// TwinCAT 3 PLC project HeatPumpTestBenchControl
// ProgramVersion: 3.1.4022.1
// CompilerDefines: VISU_USEPROPERTYINFO
// libraries:
//   VisuElem3DPath, 3.5.6.0 (System)
//   VisuElemMeter, 3.5.6.0 (System)
//   VisuElems, 3.5.6.10 (System)
//   VisuElemsDateTime, 3.5.6.0 (System)
//   VisuElemsSpecialControls, 3.5.6.0 (System)
//   VisuElemsWinControls, 3.5.6.0 (System)
//   VisuElemTextEditor, 3.5.6.0 (System)
//   visuinputs, 3.5.6.0 (system)
//   VisuNativeControl, 3.5.6.0 (System)
//   Tc2_Standard, * (Beckhoff Automation GmbH)
//   Tc2_System, * (Beckhoff Automation GmbH)
//   Tc2_Utilities, * (Beckhoff Automation GmbH)
//   Tc3_Module, * (Beckhoff Automation GmbH)
//   VisuDialogs, * (System)
// project tree:
//   DUTs/ E_PowMeas.TcDUT, E_Press.TcDUT, E_TempSensVR10.TcDUT, E_TempSensPT100.TcDUT, E_IndexPowMeas.TcDUT, E_SMStatus.TcDUT (not stored), E_TempSensVR11.TcDUT (not stored), E_Terminals.TcDUT, ST_InputVar.TcDUT, ST_InputVar_PowMeas.TcDUT, ST_OutputVar.TcDUT (not stored), ST_PumpTime.TcDUT (not stored)
//   / GlobalTextList.TcGTLO, PlcTask.TcTTO (not stored), Visualization Manager.TcVMO (not stored)
//   GVLs/ DigOutputs.TcGVL (not stored), HeatingCurve.TcGVL (not stored), AnaOutputs.TcGVL, PID.TcGVL (not stored), PowMeas.TcGVL, Pressures.TcGVL, PumpTiming.TcGVL (not stored), StateMachine.TcGVL, SysCheck.TcGVL (not stored), SysCheckParams.TcGVL (not stored), TempConvDat.TcGVL (not stored), Temperatures.TcGVL (not stored), TempSetpoints.TcGVL (not stored), TerminalErrorRT.TcGVL (not stored), TimeProgs.TcGVL (not stored)
//   POUs/ CheckDivDInt.TcPOU (not stored), CheckDivLInt.TcPOU, CheckDivLReal.TcPOU, CheckDivReal.TcPOU (not stored), MAIN.TcPOU, P_GetTime.TcPOU
//   POUs/Control/ FB_AuxHeatCont.TcPOU, FB_CyclingControl.TcPOU (not stored), P_ControlMain.TcPOU
//   POUs/Control/TemperatureControl/ FB_PIDSuppTemp.TcPOU (not stored), FB_SimpleTempCont.TcPOU (not stored), F_GetTempSP.TcPOU, I_TempController.TcIO, P_SHSuppTempPID.TcPOU (not stored)
//   POUs/ErrorHandling/ F_WriteErrLog.TcPOU, P_EmShutdownAll.TcPOU, P_EmShutdownBPumpRun.TcPOU (not stored), P_EmShutdownHCPumpRun.TcPOU, P_EmShutdownPumpsRun.TcPOU, P_EmShutdownMain.TcPOU, P_ErrorHandlingMain.TcPOU, P_WriteErrLog.TcPOU
//   POUs/Initialize/ FB_InitPumpTimes.TcPOU (not stored), FB_ReadHeatCurve.TcPOU, FB_ReadNightMode.TcPOU, FB_ReadPressTab.TcPOU, FB_ReadPT100Tab.TcPOU, FB_ReadTempResTabVR11.TcPOU, P_InitMain.TcPOU (not stored), FB_ReadTempResTabVR10.TcPOU, FB_InitTimes.TcPOU
//   POUs/Read/ F_LinSens.TcPOU (not stored), F_NTCSens.TcPOU, F_PowMeasPhase.TcPOU, P_PowMeas.TcPOU (not stored), P_ReadMain.TcPOU (not stored), P_TestVals.TcPOU
//   POUs/SystemCheck/ F_CheckAmbTemp.TcPOU, F_CheckBrinePressure.TcPOU, F_CheckCompCycPress.TcPOU (not stored), F_CheckCompOutTemp.TcPOU (not stored), F_CheckHeatCirPress.TcPOU (not stored), F_CheckHeatCirTemp.TcPOU, F_CheckPhaseSeq.TcPOU, F_CheckSens.TcPOU, F_CheckTerm.TcPOU, P_SysCheckMain.TcPOU (not stored)
//   POUs/Write/ F_ConvLinAnaOutp.TcPOU, F_PumpConvPercVolt.TcPOU, FB_RampPump.TcPOU, P_WriteMain.TcPOU (not stored)
//   VISUs/ Vis_ManCont.TcVIS (not stored), StandardVis.TcVIS
// real-time tasks:
//   TASK PlcTask: cycle T#10ms, priority 20, ADS port 350
// I/O:
//   DEVICE Device 1 (EtherCAT) (disabled), AmsNetId 134.61.132.51.2.1
//     Coupler (EK1100) [EK1100 EtherCAT Coupler (2A E-Bus)]
//       InpPressSens (EL3064) [EL3064 4Ch. Ana. Input 0-10V]
//       InpTempSens1 (EL3204-0200) [EL3204-0200 4Ch. Ana. In. PT1000 (RTD)]
//       InpTempSens2 (EL3204-0200) [EL3204-0200 4Ch. Ana. In. PT1000 (RTD)]
//       InpTempSens3 (EL3204-0200) [EL3204-0200 4Ch. Ana. In. PT1000 (RTD)]
//       InpPowMeas (EL3403-0010) [EL3403-0010 3Ch. Power Measuring, 5A]
//       AnalogOutp (EL4004) [EL4004 4Ch. Ana. Output 0-10V, 12bit]
//       OutpSwitchValv (EL2652) [EL2652 2Ch. Relay Output, CO (230V AC / 30V DC)]
//       OutpCont (EL2622) [EL2622 2Ch. Relay Output, NO (230V AC / 30V DC)]
//       InpTempSens3wire (EL3214) [EL3214 4Ch. Ana. Input PT100 (RTD)]

// ---- DUTs/E_PowMeas.TcDUT
TYPE E_PowMeas :
(
	L1,	//power phase 1
	L2,	//power phase 2
	L3	//power phase 3
);
END_TYPE

// ---- DUTs/E_Press.TcDUT
TYPE E_Press :
(
	HP,		//High pressure - after compression
	LP,		//Low pressure	- before compression
	HCP,	//Heating circuit pressure
	BP		//Brine circuit pressure
);
END_TYPE

// ---- DUTs/E_TempSensVR10.TcDUT
TYPE E_TempSensVR10 : //all VR10 temperature sensors
(
	SP,		//Temperature of DHW storage tank
	VF1,	//Temperature at the top of the space heating buffer tank
	VF2,	//Temperature after external mixing valve
	RF1		//Temperature at the bottom of the space heating buffer tank
);
END_TYPE

// ---- DUTs/E_TempSensPT100.TcDUT
TYPE E_TempSensPT100 :
(
	TExpVEv,	//Temperature between expansion valve and evaporator
	TShEv,		//Temperature after evaporator
	TCond,		//Temperature after condenser
	TAmb		//Ambient temperature
);
END_TYPE

// ---- DUTs/E_IndexPowMeas.TcDUT
TYPE E_IndexPowMeas :
//Index-value connection of the second output of the power measurement terminal
(ApparantPower, ReactivePower, Energy, cosPhi, Frequency, negEnergy);
END_TYPE

// ---- DUTs/E_Terminals.TcDUT
TYPE E_Terminals :
(
	TempSens1,
	TempSens2,
	TempSens3,
	TempSens3Wire,
	PressSens,
	PowMeasTerm,
	AnalogOutp,
	OutpSwitchValv,
	OutpCont
);
END_TYPE

// ---- DUTs/ST_InputVar.TcDUT
TYPE ST_InputVar :
STRUCT
	(*
fVar = nVarInput*fParaM + fParaC

fParaMinVal<=fVal<=fParaMaxVal
	*)	
	
	//Raw input from terminal
	nVarInput	AT %I*	:DINT; 		//Integer input from terminal
	bSensErr	AT %I*	:BOOL;		//Sensor error bit
	
	//Physical value
	fVal				:REAL;		//Input value as REAL/FLOAT/SINGLE
	
	//Linear conversion factors
	fParaM				:REAL; 		//slope of linear conversion
	fParaC				:REAL;		//offset of linear conversion
	
	//Physical limits
	fParaMaxVal			:REAL;		//Maximum physical value
	fParaMinVal			:REAL;		//Minimum physical value
	
	bValid				:BOOL	:=	TRUE;	//Indicator if fVal is valid
	
END_STRUCT
END_TYPE

// ---- DUTs/ST_InputVar_PowMeas.TcDUT
TYPE ST_InputVar_PowMeas :
STRUCT
	//Input from terminal as INT32
	nCurrentRaw	AT	%I*	:	DINT;
	nVoltRaw	AT	%I*	:	DINT;
	nEffPowRaw	AT	%I*	:	DINT;
	nVariantRaw	AT	%I*	:	DINT;				//set to cos(phi)
(*
variant input is controlled by index output:
0	-	Apparent power
1	-	Reactive power
2	-	Energy
3	-	cos(phi)
4	-	Frequency
5	-	Negative Energy
*)	
	//Index output to terminal
	nIndexOut	AT	%Q*	:	USINT	:=	3;		//cos(phi)
	
	//Physical values
	fCurrent	:	REAL;
	fVolt		:	REAL;
	fEffPow		:	REAL;
	fcosPhi		:	REAL;
	
	//Conversion factors
	fScaleCurr		:	REAL	:=	0.000005;	//Current = 0.000005A * current transformer ratio * raw value
	fScaleVolt		:	REAL	:=	0.0001;		//Voltage = 0.0001V * voltage transformer ratio * raw value
	fScaleEffPow	:	REAL	:=	0.01;		//EffPow = 0.01W * current and voltage transformer ratio
	fCurrTrans		:	REAL	:=	0.1; 		//current transformer ratio: A50/A5
	fScaleAppPow	:	REAL	:=	0.01;		//AppPow = 0.01W * current and voltage transformer ratio * raw value
	fScaleReaPow	:	REAL	:=	0.01;		//ReaPow = 0.01VAr * current and voltage transformer ratio * raw value
	fScaleEn		:	REAL	:=	0.001;		//Energy = 0.001Wh * current and voltage transformer ratio * raw value
	fScaleCosPhi	:	REAL	:=	0.001;		//CosPhi = 0.001 * raw value
	fScaleFrequ		:	REAL	:=	0.1;		//Frequ = 0.1Hz * raw value
		
END_STRUCT
END_TYPE

// ---- GVLs/AnaOutputs.TcGVL
{attribute 'qualified_only'}
VAR_GLOBAL
	stOutpBP		:	ST_OutputVar;	//Control signal for brine pump
	stOutpIntHP		:	ST_OutputVar;	//Control signal for internal heating circuit pump
	stOutpExtHP		:	ST_OutputVar;	//Control signal for external heating circuit pump
	stOutpMixValv	:	ST_OutputVar;	//Control signal for circulating pump
END_VAR

// ---- GVLs/PowMeas.TcGVL
VAR_GLOBAL
	//Power measurement values for all phases
	ePowMeas	:	E_PowMeas;
	stPowMeas	:	ARRAY[0..2]	OF ST_InputVar_PowMeas;
	
	//accumulated values
	fEffPow		:	REAL;	//Total effective power = sum of effective power of phases
	fMeanCosPhi	:	REAL;	//Mean power factor
	fAppPow		:	REAL;	//Total apparent power
	fReaPow		:	REAL;	//Total reactive power
	
	//phase sequence
	bPhaseSeq	AT	%I*	: BOOL;	//Phase sequence detected by the power measurement terminal
	//0 - Sequence L1-L3-L2 detected -> counter-clockwise net
	//1 - Sequence L1-L2-L3 detected -> clockwise net, or at least 1 wire not connected
	
END_VAR

// ---- GVLs/Pressures.TcGVL
{attribute 'qualified_only'}
VAR_GLOBAL
	ePress	:	E_Press;
	stPress	:	ARRAY[0..3] OF ST_InputVar;

(*
	stHP	:	ST_InputVar;	//High pressure - after compression
	stLP	: 	ST_InputVar;	//Low pressure	- before compression
	stHCP	:	ST_InputVar;	//Heating circuit pressure
	stBP	:	ST_InputVar;	//Brine circuit pressure
*)
END_VAR

// ---- GVLs/StateMachine.TcGVL
{attribute 'qualified_only'}
VAR_GLOBAL
	eStatus			:	E_SMStatus	:= Initialize;
	dtCurTime		:	DT;
	todCurTime		:	TOD;
	bActAuxHeat		:	BOOL	:= TRUE;	//Activate auxiliary heater
	//Fault status
	bFault			:	BOOL	:= FALSE;	//system fault indicator
	nFault			:	USINT;				//fault number
	sFaultMess		:	STRING	:= '';		//fault message
	nErrCount		:	INT		:= 0;		//error counter
	bPermShut		:	BOOL	:= FALSE;	//permanent shutdown
	bTempShut		:	BOOL	:= FALSE;	//temporary shutdown
	bEmOpPoss		:	BOOL	:= FALSE;	//emergency operation possible
	bEmOpAct		:	BOOL	:= FALSE;	//emergency operation active
	bManEmShutdown	:	BOOL	:= FALSE;	//manual emergency shutdown
	//Cycling control
	dtLastStart		:	DT;					//date and time of last start
	dtLastStop		:	DT;					//date and time of last stop
	nNumStart		:	USINT	:= 0;		//number of starts per hour
	//Control signals
	bCompRun		:	BOOL;
	bAuxHeatOp		:	BOOL;
	bSwitchVal		:	BOOL;				//True: space heating mode || False: DHW mode
	fMixVal			:	REAL;				//mixing valve position [0..10V]
	bBrinePump		:	BOOL;
	nBrinePump		:	USINT	:= 100;		//brine pump rpm in percent (0% - minimum speed, 100% - maximum speed)
	bIntHeatCPump	:	BOOL;
	nIntHeatCPump	:	USINT	:= 100;		//internal heating circuit pump rpm in percent (0% - minimum speed, 100% - maximum speed)
	bExtHeatCPump	:	BOOL;
	nExtHeatCPump	:	USINT	:= 100;		//external heating circuit pump rpm in percent (0% - minimum speed, 100% - maximum speed)
	bCircPump		:	BOOL;
END_VAR

// ---- POUs/Control/TemperatureControl/I_TempController.TcIO
INTERFACE I_TempController

//request compressor operation

//Switching valve mode: 
//True: space heating mode
//False: DHW mode

PROPERTY CompOp : BOOL
GET
END_GET
SET
END_SET
END_PROPERTY

PROPERTY SpaceHeatTempSP : REAL
GET
END_GET
SET
END_SET
END_PROPERTY

PROPERTY ValveMode : BOOL
GET
END_GET
SET
END_SET
END_PROPERTY

END_INTERFACE

// ---- POUs/CheckDivLInt.TcPOU
// Implicitly generated code : DO NOT EDIT
FUNCTION CheckDivLInt : LINT
VAR_INPUT
	divisor:LINT;
END_VAR

// Implicitly generated code : Only an Implementation suggestion
IF divisor = 0 THEN
	CheckDivLInt:=1;
	StateMachine.bFault		:=	TRUE;
	StateMachine.nFault		:=	2;
	StateMachine.sFaultMess	:=	'Critical program error: division by 0';
	StateMachine.eStatus	:=	Error;
	P_EmShutdownAll();	//Execute emergency shutdown
ELSE
	CheckDivLInt:=divisor;
END_IF;

END_FUNCTION

// ---- POUs/ErrorHandling/P_EmShutdownAll.TcPOU
PROGRAM P_EmShutdownAll
VAR
END_VAR

//shut down all components

StateMachine.bCompRun		:=	FALSE;
DigOutputs.bOutpComp		:=	FALSE;

StateMachine.bAuxHeatOp		:=	FALSE;
DigOutputs.bOutpAH			:=	FALSE;

StateMachine.bBrinePump		:=	FALSE;
AnaOutputs.stOutpBP.fVal	:=	0.75;	//0.75 Volt: Pump stop
AnaOutputs.stOutpBP			:=	F_ConvLinAnaOutp(stOutput:=AnaOutputs.stOutpBP);

StateMachine.bIntHeatCPump	:=	FALSE;
AnaOutputs.stOutpIntHP.fVal	:=	0.75;	//0.75 Volt: Pump stop
AnaOutputs.stOutpIntHP		:=	F_ConvLinAnaOutp(stOutput:=AnaOutputs.stOutpIntHP);

StateMachine.bExtHeatCPump	:=	FALSE;
AnaOutputs.stOutpExtHP.fVal	:=	0.75;	//0.75 Volt: Pump stop
AnaOutputs.stOutpExtHP			:=	F_ConvLinAnaOutp(stOutput:=AnaOutputs.stOutpExtHP);

StateMachine.bCircPump		:=	FALSE;

END_PROGRAM

// ---- POUs/Write/F_ConvLinAnaOutp.TcPOU
FUNCTION F_ConvLinAnaOutp : ST_OutputVar
VAR_INPUT
	stOutput	:	ST_OutputVar;
END_VAR
VAR
END_VAR

//nVarOutput = (fVar-fParaC)/fParaM)
stOutput.nVarOutput	:=	REAL_TO_INT((stOutput.fVal - stOutput.fParaC)*stOutput.fParaMaxOutp/stOutput.nParaMaxInt);

//assign output
F_ConvLinAnaOutp	:=	stOutput;

END_FUNCTION

// ---- POUs/CheckDivLReal.TcPOU
// Implicitly generated code : DO NOT EDIT
FUNCTION CheckDivLReal : LREAL
VAR_INPUT
	divisor:LREAL;
END_VAR

// Implicitly generated code : Only an Implementation suggestion
IF divisor = 0 THEN
	CheckDivLReal:=1;
	StateMachine.bFault		:=	TRUE;
	StateMachine.nFault		:=	2;
	StateMachine.sFaultMess	:=	'Critical program error: division by 0';
	StateMachine.eStatus	:=	Error;
	P_EmShutdownAll();	//Execute emergency shutdown
ELSE
	CheckDivLReal:=divisor;
END_IF;

END_FUNCTION

// ---- POUs/Control/FB_AuxHeatCont.TcPOU
FUNCTION_BLOCK FB_AuxHeatCont
VAR_INPUT
	bCompOp			:	BOOL	:=	FALSE; //has the controller requested compressor operation
	bCycContOK		:	BOOL; //has the cycling control authorized the compressor start-up
	bCompStart		:	BOOL; //is compressor start-up procedure active
END_VAR
VAR_OUTPUT
	bAuxHeatOp	:	BOOL;
END_VAR
VAR
	eVF1	:	E_TempSensVR10	:=	VF1;
	eSP		:	E_TempSensVR10	:=	SP;
	SampTim	:	TON();						//Sampling timer
	fBuffVF1:	ARRAY[0..nAuxHeatStart] OF REAL;	//Buffer
	fBuffSP	:	ARRAY[0..nAuxHeatStart] OF REAL;	//Buffer
	i		:	INT;
	bAuxCap	:	BOOL;
END_VAR
VAR CONSTANT
	nAuxHeatStart	:	INT		:=	180;	//Time in seconds the auxiliary heater control waits for the heat pump to be effective
END_VAR

IF bCompOp AND (NOT bAuxHeatOp) AND bCycContOK THEN

	SampTim.IN	:=	TRUE;
	SampTim.PT	:=	T#1s;
	SampTim();

	IF SampTim.Q THEN
		FOR i := 0 TO nAuxHeatStart - 1 DO
			fBuffVF1[i]	:=	fBuffVF1[i+1];
		END_FOR
		fBuffVF1[nAuxHeatStart] := Temperatures.stTempSensVR10[eVF1].fVal; //save current temperature in buffer
	
		FOR i := 0 TO nAuxHeatStart - 1 DO
			fBuffSP[i]	:=	fBuffSP[i+1];
		END_FOR
		fBuffSP[nAuxHeatStart] := Temperatures.stTempSensVR10[eSP].fVal; //save current temperature in buffer
	
		//reset timer
		SampTim.IN	:=	FALSE;
		SampTim();
	END_IF
	
	//check if auxiliary heater is needed
	IF StateMachine.bSwitchVal THEN	//space heating mode
		IF (fBuffVF1[nAuxHeatStart] < fBuffVF1[0]) THEN //temperature in buffer tank has not increased
			bAuxHeatOp	:=	TRUE;	//activate auxiliary heater
			bAuxCap		:=	TRUE;
		END_IF
	ELSE	//DHW mode
		IF (fBuffSP[nAuxHeatStart] < fBuffSP[0]) THEN //temperature in buffer tank has not increased
			bAuxHeatOp	:=	TRUE;	//activate auxiliary heater
			bAuxCap		:=	TRUE;
		END_IF
	END_IF
ELSIF bCompOp AND  (NOT bAuxHeatOp) AND (NOT bCycContOK) THEN	//heat demand, but compressor cannot start
	bAuxHeatOp	:=	TRUE;	
ELSIF (NOT bCompOp) THEN	//deactivate auxiliary heater when no compressor operation is needed
	bAuxHeatOp	:=	FALSE;
	bAuxCap 	:=	FALSE;
ELSIF bAuxHeatOp AND bCycContOK AND (NOT bAuxCap) AND NOT (bCompStart) THEN //deactivate auxiliary heater when the compressor can start again
	bAuxHeatOp := FALSE;
END_IF

END_FUNCTION_BLOCK

// ---- POUs/Control/P_ControlMain.TcPOU
PROGRAM P_ControlMain
VAR_INPUT
	bEmOp				:	BOOL	:=	FALSE;	//Emergency operation
END_VAR
VAR
	iTempCont			:	I_TempController;	//temperature controller interface
	//function block instances
	fbSimpleTempCont	:	FB_SimpleTempCont;	//temperature controller
	fbCycCont			:	FB_CyclingControl;
	fbAuxHeatCont		:	FB_AuxHeatCont;		//auxiliary heater control
	
	//compressor startup and shutdown flags
	bCompStart				:	BOOL	:= FALSE;
	bCompStop				:	BOOL	:= FALSE;
	bShutdownPump			:	BOOL	:= FALSE;
	bShutdownPumpAux		:	BOOL;
	bAuxHeatOld				:	BOOL;
	
	//pump timing
	TimBP					:	TON;
	TimIntHeatCir			:	TON;
	TimIntHeatCirAux		:	TON;
	TimIntHeatCirEm			:	TON;
END_VAR

//These lines need to be adjusted to use a different controller
fbSimpleTempCont();					//execute temperature control function block
iTempCont	:=	fbSimpleTempCont;	//assign function block to interface

//set switching valve mode
StateMachine.bSwitchVal	:=	iTempCont.ValveMode;

//read space heating temperature setpoint
TempSetpoints.fSpaceHeatSP	:=	iTempCont.SpaceHeatTempSP;

IF (NOT bEmOp) THEN //normal operation
	
	//operate circulating pump
	IF (TOD_TO_DINT(StateMachine.todCurTime) > TOD_TO_DINT(TimeProgs.todNightModeEnd)) AND
		(TOD_TO_DINT(StateMachine.todCurTime) < TOD_TO_DINT(TimeProgs.todNightModeStart)) THEN //day
		StateMachine.bCircPump	:=	TRUE;
	ELSE
		StateMachine.bCircPump	:=	FALSE;
	END_IF

	IF iTempCont.CompOp AND (NOT StateMachine.bCompRun) THEN	//compressor operation requested by controller and compressor not already running
		//execute cycling control
		fbCycCont();
		IF (NOT StateMachine.bFault) AND fbCycCont.bStartupOK THEN	//system is not in fault state and cycling OK
			bCompStart	:=	TRUE;		//give compressor start signal
		END_IF
	ELSIF (NOT iTempCont.CompOp) AND StateMachine.bCompRun THEN	//no compressor operation requested by controller and compressor running
		//execute cycling control
		fbCycCont();
		IF fbCycCont.bShutdownOK THEN
			bCompStop	:= TRUE;
		END_IF
	END_IF

	//compressor startup procedure
	IF bCompStart THEN
		//start pumps
		IF PumpTiming.stBPTime.bFirst THEN					//brine pump first
			StateMachine.bBrinePump	:=	TRUE;
			TimBP.PT				:=	PumpTiming.stBPTime.tPre;
			TimBP.IN				:=	TRUE;
			TimIntHeatCir.PT		:=	PumpTiming.stIntHeatCirTime.tDelay;
			TimIntHeatCir.IN		:=	TRUE;
			TimBP();
			TimIntHeatCir();
			IF TimIntHeatCir.Q THEN
				StateMachine.bIntHeatCPump	:=	TRUE;
			END_IF
		ELSIF PumpTiming.stIntHeatCirTime.bFirst THEN		//internal heating circuit pump first
			StateMachine.bIntHeatCPump	:=	TRUE;
			TimIntHeatCir.PT			:=	PumpTiming.stIntHeatCirTime.tPre;
			TimIntHeatCir.IN			:=	TRUE;
			TimBP.PT					:=	PumpTiming.stBPTime.tDelay;
			TimBP.IN					:=	TRUE;
			TimIntHeatCir();
			TimBP();
			IF TimBP.Q THEN
				StateMachine.bBrinePump		:=	TRUE;
			END_IF
		END_IF
	
		//start compressor
		IF TimBP.Q AND TimIntHeatCir.Q THEN
			//reset timers
			TimBP.IN					:=	FALSE;
			TimIntHeatCir.IN			:=	FALSE;
			TimBP();
			TimIntHeatCir();
		
			StateMachine.dtLastStart	:=	StateMachine.dtCurTime;
			StateMachine.nNumStart		:=	StateMachine.nNumStart + 1;	//startup counter
			StateMachine.bCompRun		:=	TRUE;
			bCompStart					:=	FALSE;						//startup complete
		END_IF
	END_IF

	//compressor shutdown procedure
	IF bCompStop THEN
		StateMachine.dtLastStop		:=	StateMachine.dtCurTime;
		StateMachine.bCompRun		:=	FALSE;
		bShutdownPump				:=	TRUE;
		bCompStop					:=	FALSE;
	END_IF

	IF bShutDownPump THEN
		//pump timing
		TimBP.PT					:=	PumpTiming.stBPTime.tPost;
		TimBP.IN					:=	TRUE;
		TimIntHeatCir.PT			:=	PumpTiming.stIntHeatCirTime.tPost;
		TimIntHeatCir.IN			:=	TRUE;
		TimBP();
		TimIntHeatCir();
		IF TimBP.Q THEN	//stop brine pump
			TimBP.IN				:=	FALSE;
			StateMachine.bBrinePump	:=	FALSE;
		END_IF
		IF TimIntHeatCir.Q THEN	//stop internal heating circuit pump
			TimIntHeatCir.IN			:=	FALSE;
			StateMachine.bIntHeatCPump	:=	FALSE;
		END_IF
		IF TimIntHeatCir.Q AND TimBP.Q THEN
			TimBP();
			TimIntHeatCir();
			bShutDownPump				:=	FALSE;	//shutdown complete
		END_IF
	END_IF
	TimIntHeatCirEm(IN:=FALSE); //reset emergency operation timer
ELSE	//emergency operation
	StateMachine.bCompRun		:=	FALSE;
	StateMachine.bBrinePump		:=	FALSE;
	StateMachine.bIntHeatCPump	:=	TRUE;
	TimIntHeatCirEm(IN:=TRUE,PT:=PumpTiming.stIntHeatCirTime.tPre);
	StateMachine.bCircPump		:=	TRUE;
	IF iTempCont.CompOp AND TimIntHeatCirEm.Q THEN	//start auxiliary heater if temperature controller identifies demand
		StateMachine.bAuxHeatOp	:=	TRUE;
	ELSE
		StateMachine.bAuxHeatOp	:=	FALSE;
	END_IF
END_IF

//space heating supply temperature and external heating circuit pump control
P_SHSuppTempPID();

//regular auxiliary heater control
IF NOT bEmOp THEN
	IF StateMachine.bActAuxHeat THEN
		fbAuxHeatCont(bCompOp:=iTempCont.CompOp, bCycContOK:=fbCycCont.bStartupOK, bCompStart:=bCompStart);
		IF fbAuxHeatCont.bAuxHeatOp THEN			//auxiliary heater operation requested
			StateMachine.bIntHeatCPump	:=	TRUE;	//start internal heating circuit pump
			TimIntHeatCirAux(IN:=TRUE, PT:=PumpTiming.stIntHeatCirTime.tPre);
			IF TimIntHeatCirAux.Q THEN				//after 1 minute
				StateMachine.bAuxHeatOp := TRUE;	//start auxiliary heater
				TimIntHeatCirAux(In:=FALSE);		//reset timer
			END_IF
		ELSE
			StateMachine.bAuxHeatOp	:=	FALSE;
		END_IF
	ELSE
		StateMachine.bAuxHeatOp	:=	FALSE;
	END_IF
	
	IF (NOT StateMachine.bAuxHeatOp) AND bAuxHeatOld THEN	//auxiliary heater was active last cycle
		bShutdownPumpAux	:=	TRUE;
	END_IF
	
END_IF

IF bShutdownPumpAux THEN
	TimIntHeatCirAux(IN:=TRUE, PT:=PumpTiming.stIntHeatCirTime.tPost);
	IF TimIntHeatCirAux.Q THEN
		StateMachine.bIntHeatCPump	:=	FALSE;
		TimIntHeatCirAux(In:=FALSE);
		bShutdownPumpAux	:=	FALSE;
	END_IF
END_IF

bAuxHeatOld	:=	StateMachine.bAuxHeatOp;

END_PROGRAM

// ---- POUs/Control/TemperatureControl/F_GetTempSP.TcPOU
FUNCTION F_GetTempSP : REAL
VAR_INPUT
	fAmbTemp	:	REAL;	//Ambient temperature
END_VAR
VAR
	i			:	USINT	:= 0;
	nLeftInd	:	USINT;
	nRightInd	:	USINT;
	bFound		:	BOOL	:=	FALSE;	//flag if left and right element were found
	
	fDiffSet	:	REAL;				//difference between room temperature setpoint and 20°C
	fSlopeAdap	:	REAL	:=	2;		//slope of space heating setpoint adaption
	
	fIntVal		:	REAL;				//interpolated value
	fSetpoint	:	REAL;				//space heating temperature setpoint
END_VAR

FOR i:=1 TO 40 DO
	IF NOT bFound THEN
		IF HeatingCurve.HeatCurve[i,0] >= fAmbTemp THEN
			nLeftInd	:=	i - 1;
			nRightInd	:=	i;
			bFound		:=	TRUE;
		END_IF
	END_IF
END_FOR

//perform interpolation
IF bFound THEN
	fIntVal	:=	HeatingCurve.HeatCurve[nLeftInd,1] + ((HeatingCurve.HeatCurve[nRightInd,1] - HeatingCurve.HeatCurve[nLeftInd,1])/(HeatingCurve.HeatCurve[nRightInd,0] - HeatingCurve.HeatCurve[nLeftInd,0])) * (fAmbTemp - HeatingCurve.HeatCurve[nLeftInd,0]);
ELSIF HeatingCurve.HeatCurve[0,0] >= fAmbTemp THEN	//ambient temperature lower than minimum value in heating curve
	fIntVal	:=	HeatingCurve.HeatCurve[0,1];
ELSIF fAmbTemp >= HeatingCurve.HeatCurve[40,0] THEN	//ambient temperature higher than maximum value in heating curve
	fIntVal	:=	HeatingCurve.HeatCurve[40,1];
END_IF

//adapt to room temperature setpoint
IF (TOD_TO_UDINT(StateMachine.todCurTime) > TOD_TO_UDINT(TimeProgs.todNightModeEnd)) AND
	(TOD_TO_UDINT(StateMachine.todCurTime) < TOD_TO_UDINT(TimeProgs.todNightModeStart)) THEN	//day
	fDiffSet	:=	TempSetpoints.fRoomSetpoint - 20;
ELSE	//night
	fDiffSet	:=	TempSetpoints.fRoomSetpointNight - 20;
END_IF
fSetpoint	:=	fIntVal + (fDiffSet * fSlopeAdap);

//assign output
F_GetTempSP	:=	fSetpoint;

END_FUNCTION

// ---- POUs/ErrorHandling/F_WriteErrLog.TcPOU
FUNCTION F_WriteErrLog : BOOL
VAR_INPUT
END_VAR
VAR
END_VAR

END_FUNCTION

// ---- POUs/ErrorHandling/P_EmShutdownHCPumpRun.TcPOU
PROGRAM P_EmShutdownHCPumpRun
VAR
END_VAR

//shut down all components except heating circuit pumps

StateMachine.bCompRun		:=	FALSE;
DigOutputs.bOutpComp		:=	FALSE;

StateMachine.bAuxHeatOp		:=	FALSE;
DigOutputs.bOutpAH			:=	FALSE;

StateMachine.bBrinePump		:=	FALSE;
AnaOutputs.stOutpBP.fVal	:=	0.75;	//0.75 Volt: Pump stop
AnaOutputs.stOutpBP			:=	F_ConvLinAnaOutp(stOutput:=AnaOutputs.stOutpBP);

StateMachine.bIntHeatCPump	:=	TRUE;
AnaOutputs.stOutpIntHP.fVal	:=	10;
AnaOutputs.stOutpIntHP		:=	F_ConvLinAnaOutp(stOutput:=AnaOutputs.stOutpIntHP);

StateMachine.bExtHeatCPump	:=	TRUE;
AnaOutputs.stOutpExtHP.fVal	:=	10;
AnaOutputs.stOutpExtHP			:=	F_ConvLinAnaOutp(stOutput:=AnaOutputs.stOutpExtHP);

StateMachine.bCircPump		:=	TRUE;

END_PROGRAM

// ---- POUs/ErrorHandling/P_EmShutdownPumpsRun.TcPOU
PROGRAM P_EmShutdownPumpsRun
VAR
END_VAR

//shut down all components except pumps

StateMachine.bCompRun		:=	FALSE;
DigOutputs.bOutpComp		:=	FALSE;

StateMachine.bAuxHeatOp		:=	FALSE;
DigOutputs.bOutpAH			:=	FALSE;

StateMachine.bBrinePump		:=	TRUE;
AnaOutputs.stOutpBP.fVal	:=	10;
AnaOutputs.stOutpBP			:=	F_ConvLinAnaOutp(stOutput:=AnaOutputs.stOutpBP);

StateMachine.bIntHeatCPump	:=	TRUE;
AnaOutputs.stOutpIntHP.fVal	:=	10;
AnaOutputs.stOutpIntHP		:=	F_ConvLinAnaOutp(stOutput:=AnaOutputs.stOutpIntHP);

StateMachine.bExtHeatCPump	:=	TRUE;
AnaOutputs.stOutpExtHP.fVal	:=	10;
AnaOutputs.stOutpExtHP			:=	F_ConvLinAnaOutp(stOutput:=AnaOutputs.stOutpExtHP);

StateMachine.bCircPump		:=	TRUE;

END_PROGRAM

// ---- POUs/ErrorHandling/P_EmShutdownMain.TcPOU
PROGRAM P_EmShutdownMain
VAR
END_VAR

IF StateMachine.bManEmShutdown THEN
	StateMachine.bFault		:=	TRUE;
	StateMachine.nFault		:=	1;
	StateMachine.sFaultMess	:=	'Manual emergency shutdown';
END_IF

//emergency shutdown scenarios

//manual emergency shutdown or terminal communication error or initialization failed or division by 0 detected -> stop all components
IF StateMachine.bManEmShutdown OR SysCheck.bTermErrRT OR (StateMachine.nFault = 10) OR (StateMachine.nFault = 2) THEN
	P_EmShutdownAll();	//complete shutdown	
//only brine pressure fault -> keep heating circuit pump running
ELSIF (SysCheck.bBP OR (StateMachine.nFault = 54)) AND (NOT SysCheck.bHCP) THEN //brine pressure too low or sensor failure
	P_EmShutdownHCPumpRun();
//only heating circuit pressure fault -> keep brine pump running
ELSIF (SysCheck.bHCP OR (StateMachine.nFault = 53)) AND (NOT SysCheck.bBP) THEN //heating circuit pressure too low or sensor failure
	P_EmShutdownBPumpRun();
//other faults keep all pumps running
ELSE
	P_EmShutdownPumpsRun();
END_IF

END_PROGRAM

// ---- POUs/ErrorHandling/P_ErrorHandlingMain.TcPOU
PROGRAM P_ErrorHandlingMain
VAR
	HCPTim	:	TON;
	BPTim	:	TON;
END_VAR

//error handling for each fault that can occur
CASE StateMachine.nFault OF
	
	1:	//manual emergency shutdown
		StateMachine.bPermShut	:=	TRUE;
		StateMachine.bEmOpPoss	:=	FALSE;
		
	2:	//division by 0
		StateMachine.bPermShut	:=	TRUE;
		StateMachine.bEmOpPoss	:=	FALSE;
		
	10:	//Initialization failed
		StateMachine.bPermShut	:=	TRUE;
		StateMachine.bEmOpPoss	:=	FALSE;

	21:	//compressor outlet temperature too high
		StateMachine.bTempShut	:=	TRUE;	//wait for a lower temperature
		IF NOT SysCheck.bHCP THEN	//enable emergency operation if heating circuit pressure is ok
			StateMachine.bEmOpPoss	:=	TRUE;
		END_IF

	31, 32:	//heating circuit temperatures too high
		StateMachine.bTempShut	:=	TRUE;	//wait for lower temperatures
		StateMachine.bEmOpPoss	:=	FALSE;
		
	41, 42:	//ambient temperature too high or low
		StateMachine.bTempShut	:=	TRUE;	//wait for a suitable ambient temperature
		IF NOT SysCheck.bHCP THEN	//enable emergency operation if heating circuit pressure is ok
			StateMachine.bEmOpPoss	:=	TRUE;
		END_IF

	43:	//brine pressure too low
		StateMachine.bTempShut	:=	TRUE;
		IF NOT SysCheck.bHCP THEN	//enable emergency operation if heating circuit pressure is ok
			StateMachine.bEmOpPoss	:=	TRUE;
		END_IF
		BPTim.PT				:=	T#5M;
		BPTim.IN				:=	TRUE;
		BPTim();
		IF BPTim.Q THEN	//if the brine circuit pressure stays too low for 5 mins, switch to permanent shutdown
			StateMachine.bTempShut	:=	FALSE;
			StateMachine.bPermShut	:=	TRUE;
			BPTim.IN				:=	FALSE;
			BPTim();
		END_IF

	44:	//heating circuit pressure too low
		StateMachine.bTempShut	:=	TRUE;
		StateMachine.bEmOpPoss	:=	FALSE;
		HCPTim.PT				:=	T#5M;
		HCPTim.IN				:=	TRUE;
		HCPTim();
		IF HCPTim.Q THEN	//if the heating circuit pressure stays too low for 5 mins, switch to permanent shutdown
			StateMachine.bTempShut	:=	FALSE;
			StateMachine.bPermShut	:=	TRUE;
			HCPTim.IN				:=	FALSE;
			HCPTim();
		END_IF
		
	45, 46:	//evaporation pressure too low or condensation pressure too high
		StateMachine.bTempShut	:=	TRUE;
		IF NOT SysCheck.bHCP THEN	//enable emergency operation if heating circuit pressure is ok
			StateMachine.bEmOpPoss	:=	TRUE;
		END_IF

	47:	//phase sequence error
		StateMachine.bPermShut	:=	TRUE;
		IF NOT SysCheck.bHCP THEN	//enable emergency operation if heating circuit pressure is ok
			StateMachine.bEmOpPoss	:=	TRUE;
		END_IF
		
	51, 52, 54: //brine circuit pressure, high pressure or low pressure sensor failure
		StateMachine.bPermShut	:=	TRUE;
		IF NOT SysCheck.bHCP THEN	//enable emergency operation if heating circuit pressure is ok
			StateMachine.bEmOpPoss	:=	TRUE;
		END_IF
		
	53:	//heating circuit pressure sensor failure
		StateMachine.bPermShut	:=	TRUE;
		StateMachine.bEmOpPoss	:=	FALSE;	//disable emergency operation in case heating circuit pressure is too low
		
	64:	//ambient temperature sensor failure
		StateMachine.bPermShut	:=	TRUE;
		IF NOT SysCheck.bHCP THEN	//enable emergency operation if heating circuit pressure is ok
			StateMachine.bEmOpPoss	:=	TRUE;
		END_IF	
		
	71, 72, 73, 74, 75, 76, 77, 78:	//internal temperature sensor failure
		StateMachine.bPermShut	:=	TRUE;
		IF NOT SysCheck.bHCP THEN	//enable emergency operation if heating circuit pressure is ok
			StateMachine.bEmOpPoss	:=	TRUE;
		END_IF
		
	81, 82, 83, 84:	//external temperature sensor failure
		StateMachine.bPermShut	:=	TRUE;
		StateMachine.bEmOpPoss	:=	FALSE; //disable emergency operation to prevent dangerous temperatures
		
	91, 92, 93, 94, 95, 96, 97, 98, 99:	//real-time communication failure
		StateMachine.bPermShut	:=	TRUE;
		StateMachine.bEmOpPoss	:=	FALSE;

END_CASE

END_PROGRAM

// ---- POUs/ErrorHandling/P_WriteErrLog.TcPOU
PROGRAM P_WriteErrLog
VAR_INPUT
	bStart		:	BOOL;
END_VAR
VAR
	nStep		:	USINT;

	fbFileOpen	:	FB_FileOpen;
	fbFileClose	:	FB_FileClose;
	sErrLogPath	:	STRING	:=	'D:\cve-mme\WpPruefstandData\ErrorLog.txt';
	
	fbFilePuts	:	FB_FilePuts;
	sErrLogMess	:	STRING;
	
	hLogFile	:	UINT;
	nErrCount	:	INT		:=	0;
END_VAR

CASE nStep OF
	
	0:	//idle
		IF bStart THEN
			bStart	:=	FALSE;
			nStep	:=	1;
		END_IF

	1:	//open ErrorLog File
		fbFileOpen(sNetId:='', sPathName:=sErrLogPath, nMode:=FOPEN_MODEAPPEND OR FOPEN_MODEPLUS, bExecute:=TRUE);
		nStep	:=	2;
		
	2:
		IF fbFileOpen.bError THEN
			nStep	:=	0;
		END_IF
		
		IF fbFileOpen.bBusy THEN
			fbFileOpen(bExecute:=FALSE);
		ELSE
			fbFileOpen(bExecute:=FALSE);
			hLogFile	:=	fbFileOpen.hFile;
			sErrLogMess	:=	CONCAT(str1:=DT_TO_STRING(StateMachine.dtCurTime),
				str2:=CONCAT(str1:='$t',str2:=CONCAT(str1:=StateMachine.sFaultMess,str2:='$n')));
			nStep		:=	3;	
		END_IF	
		
	3:	//write data
		fbFilePuts(sNetId:='',hFile:=hLogFile,sLine:=sErrLogMess,bExecute:=TRUE);
		nStep			:=	4;
		
	4:
		IF fbFilePuts.bError THEN
			nStep	:=	0;
		END_IF
	
		IF fbFilePuts.bBusy THEN
			fbFilePuts(bExecute:=FALSE);
		ELSE
			fbFilePuts(bExecute:=FALSE);
			nStep	:=	5;
		END_IF
		
	5:	//close file
		fbFileClose(sNetId:='',hFile:=hLogFile,bExecute:=TRUE);
		nStep	:=	6;
		
	6:	
		IF fbFileClose.bError THEN
			nStep	:=	0;
		END_IF
	
		IF fbFileClose.bBusy THEN
			fbFileClose(bExecute:=FALSE);
		ELSE
			fbFileClose(bExecute:=FALSE);
			hLogFile	:=	0;
			nStep		:=	0;	//switch to idle mode
		END_IF
END_CASE

END_PROGRAM

// ---- POUs/Initialize/FB_ReadHeatCurve.TcPOU
FUNCTION_BLOCK FB_ReadHeatCurve
VAR_INPUT
	bExecute		:	BOOL	:= FALSE;
END_VAR
VAR_OUTPUT
	bCompleted		:	BOOL	:=	FALSE;
	bError			:	BOOL	:=	FALSE;
END_VAR
VAR
	fbFileOpen		:	FB_FileOpen;
	fbFileGets		:	FB_FileGets;
	fbReader		:	FB_CSVMemBufferReader;
	fbFileClose		:	FB_FileClose;
	sCSVPath		:	STRING	:=	'*\Data\HeatingCurve.csv';	//Path to csv file
	hFile			:	UINT;
	bEOF			:	BOOL	:=	FALSE;
	Step			:	DWORD	:=	0;
	sLine			:	STRING;	//Line read by fbFileGets
	nLine			:	UINT	:=	0;
END_VAR

CASE Step OF
	
0:	//Standby mode
	IF bExecute THEN
		bExecute	:=	FALSE; //reset to defaults
		hFile		:=	0;
		bEOF		:=	FALSE;
		bCompleted	:=	FALSE;
		bError		:=	FALSE;
		sLine		:=	'';
		nLine		:=	0;
		Step		:=	1; //start program
	END_IF

1:	//Open file
	fbFileOpen(sNetId:='', sPathName:=sCSVPath, nMode:=FOPEN_MODEREAD OR FOPEN_MODETEXT,
		ePath:=PATH_GENERIC, tTimeout:=T#5s, bExecute:=TRUE);
	Step	:=	Step + 1;

2:
	fbFileOpen(bExecute:=FALSE);
	IF NOT fbFileOpen.bBusy THEN
		IF NOT fbFileOpen.bError THEN
			//Store file handle
			hFile	:=	fbFileOpen.hFile;
			Step	:=	Step + 1;
		ELSE
			Step	:=	90;	
		END_IF
	END_IF

3:	//Read csv file
	fbFileGets(sNetId:='', hFile:=hFile, bExecute:=TRUE, tTimeout:=T#5S);
	nLine	:=	nLine + 1;
	Step	:=	Step + 1;

4:
	fbFileGets(bExecute:=FALSE);
	IF NOT fbFileGets.bBusy THEN
		IF NOT (nLine = 1) THEN //Header -> jump to next line
			IF NOT fbFileGets.bError THEN
				IF fbFileGets.bEOF THEN
					Step	:=	10; //Reached end of file
				ELSE
					sLine	:=	fbFileGets.sLine; //store line
					IF RIGHT(sLine,1) = '$L' THEN
						sLine	:=	REPLACE(sLINE, '$R$L', 2, LEN(sLine)); //restore CRLF characters
					END_IF
					Step	:=	Step + 1;
				END_IF
			ELSE
				Step	:=	90;
			END_IF
		ELSE
			Step	:=	3;
		END_IF
	END_IF
	
5:	//Parse line
	
	fbReader.eCmd	:=	eEnumCmd_First;	//Read first value (ambient temperature)
	fbReader(pBuffer:=ADR(sLine), cbBuffer:=SIZEOF(sLine));
	
	IF fbReader.bOk THEN
		HeatingCurve.HeatCurve[nLine-2,0] := STRING_TO_REAL(fbReader.getValue);	//account for header
	ELSE
		Step	:=	90;
	END_IF	
	
	fbReader.eCmd	:=	eEnumCmd_Next;	//Read next value (temperature setpoint)
	fbReader(pBuffer:=ADR(sLine), cbBuffer:=SIZEOF(sLine));
	
	IF fbReader.bOk THEN
		HeatingCurve.HeatCurve[nLine-2,1] := STRING_TO_REAL(fbReader.getValue); //account for header
	ELSE
		Step	:=	90;
	END_IF
	
	//Read next line
	Step	:=	3;
	
10:	//end of csv file
	IF (hFile <> 0) THEN
		Step	:=	20; //close file
	END_IF
	
20:	//close csv file
	fbFileClose(bExecute:=FALSE);
	fbFileClose(sNetId:='', hFile:=hFile, bExecute:=TRUE, tTimeout:=T#5S);
	Step	:=	21;
	
21:	
	fbFileClose(bExecute:=FALSE);
	IF NOT fbFileClose.bBusy THEN
		step	:=	0;	//Standby mode
		bCompleted	:=	TRUE;
	END_IF
	
90:	//TODO: Error handling
	bError	:=	TRUE;
	IF (hFile <> 0) THEN
		Step	:=	20;	//close file
	END_IF

END_CASE

END_FUNCTION_BLOCK

// ---- POUs/Initialize/FB_ReadNightMode.TcPOU
FUNCTION_BLOCK FB_ReadNightMode
VAR_INPUT
	bExecute		:	BOOL	:= FALSE;
END_VAR
VAR_OUTPUT
	bCompleted		:	BOOL	:=	FALSE;
	bError			:	BOOL	:=	FALSE;
END_VAR
VAR
	fbFileOpen		:	FB_FileOpen;
	fbFileGets		:	FB_FileGets;
	fbReader		:	FB_CSVMemBufferReader;
	fbFileClose		:	FB_FileClose;
	sCSVPath		:	STRING	:=	'*\Data\NightMode.csv';	//Path to csv file
	hFile			:	UINT;
	bEOF			:	BOOL	:=	FALSE;
	Step			:	DWORD	:=	0;
	sLine			:	STRING;	//Line read by fbFileGets
	nLine			:	UINT	:=	0;
	nHourStart		:	USINT;
	nHourStop		:	USINT;
	nMinStart		:	USINT;
	nMinStop		:	USINT;
	nStartTime		:	UDINT;	//Start time in ms
	nStopTime		:	UDINT;	//Stop time in ms
END_VAR

CASE Step OF
	
0:	//Standby mode
	IF bExecute THEN
		bExecute	:=	FALSE; //reset to defaults
		hFile		:=	0;
		bEOF		:=	FALSE;
		bCompleted	:=	FALSE;
		bError		:=	FALSE;
		sLine		:=	'';
		nLine		:=	0;
		Step		:=	1; //start program
	END_IF

1:	//Open file
	fbFileOpen(sNetId:='', sPathName:=sCSVPath, nMode:=FOPEN_MODEREAD OR FOPEN_MODETEXT,
		ePath:=PATH_GENERIC, tTimeout:=T#5s, bExecute:=TRUE);
	Step	:=	Step + 1;

2:
	fbFileOpen(bExecute:=FALSE);
	IF NOT fbFileOpen.bBusy THEN
		IF NOT fbFileOpen.bError THEN
			//Store file handle
			hFile	:=	fbFileOpen.hFile;
			Step	:=	Step + 1;
		ELSE
			Step	:=	90;	
		END_IF
	END_IF

3:	//Read csv file
	fbFileGets(sNetId:='', hFile:=hFile, bExecute:=TRUE, tTimeout:=T#5S);
	nLine	:=	nLine + 1;
	Step	:=	Step + 1;

4:
	fbFileGets(bExecute:=FALSE);
	IF NOT fbFileGets.bBusy THEN
		IF NOT (nLine = 1) THEN //Header -> jump to next line
			IF NOT fbFileGets.bError THEN
				IF fbFileGets.bEOF THEN
					Step	:=	10; //Reached end of file
				ELSE
					sLine	:=	fbFileGets.sLine; //store line
					IF RIGHT(sLine,1) = '$L' THEN
						sLine	:=	REPLACE(sLINE, '$R$L', 2, LEN(sLine)); //restore CRLF characters
					END_IF
					Step	:=	Step + 1;
				END_IF
			ELSE
				Step	:=	90;
			END_IF
		ELSE
			Step	:=	3;
		END_IF
	END_IF
	
5:	//Parse line
	fbReader.eCmd	:=	eEnumCmd_First;	//Read first value (identifier)
	fbReader(pBuffer:=ADR(sLine), cbBuffer:=SIZEOF(sLine));
	
	fbReader.eCmd	:=	eEnumCmd_Next;	//Read next value (hour)
	fbReader(pBuffer:=ADR(sLine), cbBuffer:=SIZEOF(sLine));
	
	IF fbReader.bOk THEN
		IF (nLine = 2) THEN
			nHourStart	:=	STRING_TO_USINT(fbReader.getValue);
		ELSIF (nLine = 3) THEN
			nHourStop	:=	STRING_TO_USINT(fbReader.getValue);
		ELSE
			Step	:=	90;
		END_IF
	ELSE
		Step	:=	90;
	END_IF	
	
	fbReader.eCmd	:=	eEnumCmd_Next;	//Read next value (minute)
	fbReader(pBuffer:=ADR(sLine), cbBuffer:=SIZEOF(sLine));
	
	IF fbReader.bOk THEN
		IF (nLine = 2) THEN
			nMinStart	:=	STRING_TO_USINT(fbReader.getValue);
		ELSIF (nLine = 3) THEN
			nMinStop	:=	STRING_TO_USINT(fbReader.getValue);
		ELSE
			Step	:=	90;
		END_IF
	ELSE
		Step	:=	90;
	END_IF
	
	//Read next line
	Step	:=	3;
	
10:	//end of csv file
	IF (hFile <> 0) THEN
		Step	:=	20; //close file
	END_IF
	
20:	//close csv file
	fbFileClose(bExecute:=FALSE);
	fbFileClose(sNetId:='', hFile:=hFile, bExecute:=TRUE, tTimeout:=T#5S);
	Step	:=	21;
	
21:	
	fbFileClose(bExecute:=FALSE);
	IF NOT fbFileClose.bBusy THEN
		//convert data and write to GVL
		nStartTime	:=	nHourStart * 3600 * 1000 + nMinStart * 60 * 1000;
		nStopTime	:=	nHourStop * 3600 * 1000 + nMinStop * 60 * 1000;
		TimeProgs.todNightModeStart	:=	UDINT_TO_TOD(nStartTime);
		TimeProgs.todNightModeEnd	:=	UDINT_TO_TOD(nStopTime);
	
		step	:=	0;	//Standby mode
		bCompleted	:=	TRUE;
	END_IF
	
90:	//TODO: Error handling
	bError	:=	TRUE;
	IF (hFile <> 0) THEN
		Step	:=	20;	//close file
	END_IF

END_CASE

END_FUNCTION_BLOCK

// ---- POUs/Initialize/FB_ReadPressTab.TcPOU
FUNCTION_BLOCK FB_ReadPressTab
VAR_INPUT
	bExecute		:	BOOL	:= FALSE;
END_VAR
VAR_OUTPUT
	bCompleted		:	BOOL	:=	FALSE;
	bError			:	BOOL	:=	FALSE;
END_VAR
VAR
	fbFileOpen		:	FB_FileOpen;
	fbFileGets		:	FB_FileGets;
	fbReader		:	FB_CSVMemBufferReader;
	fbFileClose		:	FB_FileClose;
	sCSVPath		:	STRING	:=	'*\Data\PressureDat.csv';	//Path to csv file
	hFile			:	UINT;
	bEOF			:	BOOL	:=	FALSE;
	Step			:	DWORD	:=	0;
	sLine			:	STRING;	//Line read by fbFileGets
	nLine			:	UINT	:=	0;
	nIndSens		:	INT;
	stSensName		:	String;
END_VAR

CASE Step OF
	
0:	//Standby mode
	IF bExecute THEN
		bExecute	:=	FALSE; //reset to defaults
		hFile		:=	0;
		bEOF		:=	FALSE;
		bCompleted	:=	FALSE;
		bError		:=	FALSE;
		sLine		:=	'';
		nLine		:=	0;
		Step		:=	1; //start program
	END_IF

1:	//Open file
	fbFileOpen(sNetId:='', sPathName:=sCSVPath, nMode:=FOPEN_MODEREAD OR FOPEN_MODETEXT,
		ePath:=PATH_GENERIC, tTimeout:=T#5s, bExecute:=TRUE);
	Step	:=	Step + 1;

2:
	fbFileOpen(bExecute:=FALSE);
	IF NOT fbFileOpen.bBusy THEN
		IF NOT fbFileOpen.bError THEN
			//Store file handle
			hFile	:=	fbFileOpen.hFile;
			Step	:=	Step + 1;
		ELSE
			Step	:=	90;	
		END_IF
	END_IF

3:	//Read csv file
	fbFileGets(sNetId:='', hFile:=hFile, bExecute:=TRUE, tTimeout:=T#5S);
	nLine	:=	nLine + 1;
	Step	:=	Step + 1;

4:
	fbFileGets(bExecute:=FALSE);
	IF NOT fbFileGets.bBusy THEN
		IF NOT (nLine = 1) THEN //Header -> jump to next line
			IF NOT fbFileGets.bError THEN
				IF fbFileGets.bEOF THEN
					Step	:=	10; //Reached end of file
				ELSE
					sLine	:=	fbFileGets.sLine; //store line
					IF RIGHT(sLine,1) = '$L' THEN
						sLine	:=	REPLACE(sLINE, '$R$L', 2, LEN(sLine)); //restore CRLF characters
					END_IF
					Step	:=	Step + 1;
				END_IF
			ELSE
				Step	:=	90;
			END_IF
		ELSE
			Step	:=	3;
		END_IF
	END_IF
	
5:	//Parse line
	fbReader.eCmd	:=	eEnumCmd_First;	//Read first value (identifier)
	fbReader(pBuffer:=ADR(sLine), cbBuffer:=SIZEOF(sLine));
	
	IF fbReader.bOk THEN
		stSensName	:= fbReader.getValue;	//identify index of current sensor
		IF (FIND(str1:=stSensName, str2:='HP') <> 0) THEN
			Pressures.ePress	:=	HP;
		ELSIF (FIND(str1:=stSensName, str2:='LP') <> 0) THEN
			Pressures.ePress	:=	LP;
		ELSIF (FIND(str1:=stSensName, str2:='HCP') <> 0) THEN
			Pressures.ePress	:=	HCP;
		ELSIF (FIND(str1:=stSensName, str2:='BP') <> 0) THEN
			Pressures.ePress	:=	BP;
		END_IF
		nIndSens	:=	Pressures.ePress;
	ELSE
		Step	:=	90;
	END_IF	
	
	fbReader.eCmd	:=	eEnumCmd_Next;	//Read next value (slope)
	fbReader(pBuffer:=ADR(sLine), cbBuffer:=SIZEOF(sLine));
	
	IF fbReader.bOk THEN
		Pressures.stPress[nIndSens].fParaM := STRING_TO_REAL(fbReader.getValue);
	ELSE
		Step	:=	90;
	END_IF	
	
	fbReader.eCmd	:=	eEnumCmd_Next;	//Read next value (offset)
	fbReader(pBuffer:=ADR(sLine), cbBuffer:=SIZEOF(sLine));
	
	IF fbReader.bOk THEN
		Pressures.stPress[nIndSens].fParaC := STRING_TO_REAL(fbReader.getValue); //account for header
	ELSE
		Step	:=	90;
	END_IF
	
	fbReader.eCmd	:=	eEnumCmd_Next;	//Read next value (maximum value)
	fbReader(pBuffer:=ADR(sLine), cbBuffer:=SIZEOF(sLine));
	
	IF fbReader.bOk THEN
		Pressures.stPress[nIndSens].fParaMaxVal := STRING_TO_REAL(fbReader.getValue); //account for header
	ELSE
		Step	:=	90;
	END_IF
	
	fbReader.eCmd	:=	eEnumCmd_Next;	//Read next value (minimum value)
	fbReader(pBuffer:=ADR(sLine), cbBuffer:=SIZEOF(sLine));
	
	IF fbReader.bOk THEN
		Pressures.stPress[nIndSens].fParaMinVal := STRING_TO_REAL(fbReader.getValue); //account for header
	ELSE
		Step	:=	90;
	END_IF
	
	//Read next line
	Step	:=	3;
	
10:	//end of csv file
	IF (hFile <> 0) THEN
		Step	:=	20; //close file
	END_IF
	
20:	//close csv file
	fbFileClose(bExecute:=FALSE);
	fbFileClose(sNetId:='', hFile:=hFile, bExecute:=TRUE, tTimeout:=T#5S);
	Step	:=	21;
	
21:	
	fbFileClose(bExecute:=FALSE);
	IF NOT fbFileClose.bBusy THEN
		step	:=	0;	//Standby mode
		bCompleted	:=	TRUE;
	END_IF
	
90:	//TODO: Error handling
	bError	:=	TRUE;
	IF (hFile <> 0) THEN
		Step	:=	20;	//close file
	END_IF

END_CASE

END_FUNCTION_BLOCK

// ---- POUs/Initialize/FB_ReadPT100Tab.TcPOU
FUNCTION_BLOCK FB_ReadPT100Tab
VAR_INPUT
	bExecute		:	BOOL	:= FALSE;
END_VAR
VAR_OUTPUT
	bCompleted		:	BOOL	:=	FALSE;
	bError			:	BOOL	:=	FALSE;
END_VAR
VAR
	fbFileOpen		:	FB_FileOpen;
	fbFileGets		:	FB_FileGets;
	fbReader		:	FB_CSVMemBufferReader;
	fbFileClose		:	FB_FileClose;
	sCSVPath		:	STRING	:=	'*\Data\PT100Dat.csv';	//Path to csv file
	hFile			:	UINT;
	bEOF			:	BOOL	:=	FALSE;
	Step			:	DWORD	:=	0;
	sLine			:	STRING;	//Line read by fbFileGets
	nLine			:	UINT	:=	0;
	nIndSens		:	INT;
	stSensName		:	String;
END_VAR

CASE Step OF
	
0:	//Standby mode
	IF bExecute THEN
		bExecute	:=	FALSE; //reset to defaults
		hFile		:=	0;
		bEOF		:=	FALSE;
		bCompleted	:=	FALSE;
		bError		:=	FALSE;
		sLine		:=	'';
		nLine		:=	0;
		Step		:=	1; //start program
	END_IF

1:	//Open file
	fbFileOpen(sNetId:='', sPathName:=sCSVPath, nMode:=FOPEN_MODEREAD OR FOPEN_MODETEXT,
		ePath:=PATH_GENERIC, tTimeout:=T#5s, bExecute:=TRUE);
	Step	:=	Step + 1;

2:
	fbFileOpen(bExecute:=FALSE);
	IF NOT fbFileOpen.bBusy THEN
		IF NOT fbFileOpen.bError THEN
			//Store file handle
			hFile	:=	fbFileOpen.hFile;
			Step	:=	Step + 1;
		ELSE
			Step	:=	90;	
		END_IF
	END_IF

3:	//Read csv file
	fbFileGets(sNetId:='', hFile:=hFile, bExecute:=TRUE, tTimeout:=T#5S);
	nLine	:=	nLine + 1;
	Step	:=	Step + 1;

4:
	fbFileGets(bExecute:=FALSE);
	IF NOT fbFileGets.bBusy THEN
		IF NOT (nLine = 1) THEN //Header -> jump to next line
			IF NOT fbFileGets.bError THEN
				IF fbFileGets.bEOF THEN
					Step	:=	10; //Reached end of file
				ELSE
					sLine	:=	fbFileGets.sLine; //store line
					IF RIGHT(sLine,1) = '$L' THEN
						sLine	:=	REPLACE(sLINE, '$R$L', 2, LEN(sLine)); //restore CRLF characters
					END_IF
					Step	:=	Step + 1;
				END_IF
			ELSE
				Step	:=	90;
			END_IF
		ELSE
			Step	:=	3;
		END_IF
	END_IF
	
5:	//Parse line
	fbReader.eCmd	:=	eEnumCmd_First;	//Read first value (identifier)
	fbReader(pBuffer:=ADR(sLine), cbBuffer:=SIZEOF(sLine));
	
	IF fbReader.bOk THEN
		stSensName	:= fbReader.getValue;	//identify index of current sensor
		IF (FIND(str1:=stSensName, str2:='TExpVEv') <> 0) THEN
			Temperatures.eTempSensPT100	:=	TExpVEv;
		ELSIF (FIND(str1:=stSensName, str2:='TShEv') <> 0) THEN
			Temperatures.eTempSensPT100	:=	TShEv;
		ELSIF (FIND(str1:=stSensName, str2:='TCond') <> 0) THEN
			Temperatures.eTempSensPT100	:=	TCond;
		ELSIF (FIND(str1:=stSensName, str2:='TAmb') <> 0) THEN
			Temperatures.eTempSensPT100	:=	TAmb;
		END_IF
		nIndSens	:=	Temperatures.eTempSensPT100;
	ELSE
		Step	:=	90;
	END_IF	
	
	fbReader.eCmd	:=	eEnumCmd_Next;	//Read next value (slope)
	fbReader(pBuffer:=ADR(sLine), cbBuffer:=SIZEOF(sLine));
	
	IF fbReader.bOk THEN
		Temperatures.stTempSensPT100[nIndSens].fParaM := STRING_TO_REAL(fbReader.getValue);
	ELSE
		Step	:=	90;
	END_IF	
	
	fbReader.eCmd	:=	eEnumCmd_Next;	//Read next value (offset)
	fbReader(pBuffer:=ADR(sLine), cbBuffer:=SIZEOF(sLine));
	
	IF fbReader.bOk THEN
		Temperatures.stTempSensPT100[nIndSens].fParaC := STRING_TO_REAL(fbReader.getValue); //account for header
	ELSE
		Step	:=	90;
	END_IF
	
	fbReader.eCmd	:=	eEnumCmd_Next;	//Read next value (maximum value)
	fbReader(pBuffer:=ADR(sLine), cbBuffer:=SIZEOF(sLine));
	
	IF fbReader.bOk THEN
		Temperatures.stTempSensPT100[nIndSens].fParaMaxVal := STRING_TO_REAL(fbReader.getValue); //account for header
	ELSE
		Step	:=	90;
	END_IF
	
	fbReader.eCmd	:=	eEnumCmd_Next;	//Read next value (minimum value)
	fbReader(pBuffer:=ADR(sLine), cbBuffer:=SIZEOF(sLine));
	
	IF fbReader.bOk THEN
		Temperatures.stTempSensPT100[nIndSens].fParaMinVal := STRING_TO_REAL(fbReader.getValue);
	ELSE
		Step	:=	90;
	END_IF
	
	//Read next line
	Step	:=	3;
	
10:	//end of csv file
	IF (hFile <> 0) THEN
		Step	:=	20; //close file
	END_IF
	
20:	//close csv file
	fbFileClose(bExecute:=FALSE);
	fbFileClose(sNetId:='', hFile:=hFile, bExecute:=TRUE, tTimeout:=T#5S);
	Step	:=	21;
	
21:	
	fbFileClose(bExecute:=FALSE);
	IF NOT fbFileClose.bBusy THEN
		step	:=	0;	//Standby mode
		bCompleted	:=	TRUE;
	END_IF
	
90:	//TODO: Error handling
	bError	:=	TRUE;
	IF (hFile <> 0) THEN
		Step	:=	20;	//close file
	END_IF

END_CASE

END_FUNCTION_BLOCK

// ---- POUs/Initialize/FB_ReadTempResTabVR11.TcPOU
FUNCTION_BLOCK FB_ReadTempResTabVR11
VAR_INPUT
	bExecute		:	BOOL	:= FALSE;
END_VAR
VAR_OUTPUT
	bCompleted		:	BOOL	:=	FALSE;
	bError			:	BOOL	:=	FALSE;
END_VAR
VAR
	fbFileOpen		:	FB_FileOpen;
	fbFileGets		:	FB_FileGets;
	fbReader		:	FB_CSVMemBufferReader;
	fbFileClose		:	FB_FileClose;
	sCSVPath		:	STRING	:=	'*\Data\CharacteristicVR11.csv';	//Path to csv file
	hFile			:	UINT;
	bEOF			:	BOOL	:=	FALSE;
	Step			:	DWORD	:=	0;
	sLine			:	STRING;	//Line read by fbFileGets
	nLine			:	UINT	:=	0;
END_VAR

CASE Step OF
	
0:	//Standby mode
	IF bExecute THEN
		bExecute	:=	FALSE; //reset to defaults
		hFile		:=	0;
		bEOF		:=	FALSE;
		bCompleted	:=	FALSE;
		bError		:=	FALSE;
		sLine		:=	'';
		nLine		:=	0;
		Step		:=	1; //start program
	END_IF

1:	//Open file
	fbFileOpen(sNetId:='', sPathName:=sCSVPath, nMode:=FOPEN_MODEREAD OR FOPEN_MODETEXT,
		ePath:=PATH_GENERIC, tTimeout:=T#5s, bExecute:=TRUE);
	Step	:=	Step + 1;

2:
	fbFileOpen(bExecute:=FALSE);
	IF NOT fbFileOpen.bBusy THEN
		IF NOT fbFileOpen.bError THEN
			//Store file handle
			hFile	:=	fbFileOpen.hFile;
			Step	:=	Step + 1;
		ELSE
			Step	:=	90;	
		END_IF
	END_IF

3:	//Read csv file
	fbFileGets(sNetId:='', hFile:=hFile, bExecute:=TRUE, tTimeout:=T#5S);
	nLine	:=	nLine + 1;
	Step	:=	Step + 1;

4:
	fbFileGets(bExecute:=FALSE);
	IF NOT fbFileGets.bBusy THEN
		IF NOT (nLine = 1) THEN //Header -> jump to next line
			IF NOT fbFileGets.bError THEN
				IF fbFileGets.bEOF THEN
					Step	:=	10; //Reached end of file
				ELSE
					sLine	:=	fbFileGets.sLine; //store line
					IF RIGHT(sLine,1) = '$L' THEN
						sLine	:=	REPLACE(sLINE, '$R$L', 2, LEN(sLine)); //restore CRLF characters
					END_IF
					Step	:=	Step + 1;
				END_IF
			ELSE
				Step	:=	90;
			END_IF
		ELSE
			Step	:=	3;
		END_IF
	END_IF
	
5:	//Parse line
	
	fbReader.eCmd	:=	eEnumCmd_First;	//Read first value (temperature)
	fbReader(pBuffer:=ADR(sLine), cbBuffer:=SIZEOF(sLine));
	
	IF fbReader.bOk THEN
		TempConvDat.VR11[nLine-1,2] := STRING_TO_REAL(fbReader.getValue);	//account for header
	ELSE
		Step	:=	90;
	END_IF	
	
	fbReader.eCmd	:=	eEnumCmd_Next;	//Read next value (resistance)
	fbReader(pBuffer:=ADR(sLine), cbBuffer:=SIZEOF(sLine));
	
	IF fbReader.bOk THEN
		TempConvDat.VR11[nLine-1,1] := STRING_TO_REAL(fbReader.getValue); //account for header
	ELSE
		Step	:=	90;
	END_IF
	
	//Read next line
	Step	:=	3;
	
10:	//end of csv file
	IF (hFile <> 0) THEN
		Step	:=	20; //close file
	END_IF
	
20:	//close csv file
	fbFileClose(bExecute:=FALSE);
	fbFileClose(sNetId:='', hFile:=hFile, bExecute:=TRUE, tTimeout:=T#5S);
	Step	:=	21;
	
21:	
	fbFileClose(bExecute:=FALSE);
	IF NOT fbFileClose.bBusy THEN
		step	:=	0;	//Standby mode
		bCompleted	:=	TRUE;
	END_IF
	
90:	//TODO: Error handling
	bError	:=	TRUE;
	IF (hFile <> 0) THEN
		Step	:=	20;	//close file
	END_IF

END_CASE

END_FUNCTION_BLOCK

// ---- POUs/Initialize/FB_ReadTempResTabVR10.TcPOU
FUNCTION_BLOCK FB_ReadTempResTabVR10
VAR_INPUT
	bExecute		:	BOOL	:= FALSE;
END_VAR
VAR_OUTPUT
	bCompleted		:	BOOL	:=	FALSE;
	bError			:	BOOL	:=	FALSE;
END_VAR
VAR
	fbFileOpen		:	FB_FileOpen;
	fbFileGets		:	FB_FileGets;
	fbReader		:	FB_CSVMemBufferReader;
	fbFileClose		:	FB_FileClose;
	sCSVPath		:	STRING	:=	'*\Data\CharacteristicVR10.csv';	//Path to csv file
	hFile			:	UINT;
	bEOF			:	BOOL	:=	FALSE;
	Step			:	DWORD	:=	0;
	sLine			:	STRING;	//Line read by fbFileGets
	nLine			:	UINT	:=	0;
END_VAR

CASE Step OF
	
0:	//Standby mode
	IF bExecute THEN
		bExecute	:=	FALSE; //reset to defaults
		hFile		:=	0;
		bEOF		:=	FALSE;
		bCompleted	:=	FALSE;
		bError		:=	FALSE;
		sLine		:=	'';
		nLine		:=	0;
		Step		:=	1; //start program
	END_IF

1:	//Open file
	fbFileOpen(sNetId:='', sPathName:=sCSVPath, nMode:=FOPEN_MODEREAD OR FOPEN_MODETEXT,
		ePath:=PATH_GENERIC, tTimeout:=T#5s, bExecute:=TRUE);
	Step	:=	Step + 1;

2:
	fbFileOpen(bExecute:=FALSE);
	IF NOT fbFileOpen.bBusy THEN
		IF NOT fbFileOpen.bError THEN
			//Store file handle
			hFile	:=	fbFileOpen.hFile;
			Step	:=	Step + 1;
		ELSE
			Step	:=	90;	
		END_IF
	END_IF

3:	//Read csv file
	fbFileGets(sNetId:='', hFile:=hFile, bExecute:=TRUE, tTimeout:=T#5S);
	nLine	:=	nLine + 1;
	Step	:=	Step + 1;

4:
	fbFileGets(bExecute:=FALSE);
	IF NOT fbFileGets.bBusy THEN
		IF NOT (nLine = 1) THEN //Header -> jump to next line
			IF NOT fbFileGets.bError THEN
				IF fbFileGets.bEOF THEN
					Step	:=	10; //Reached end of file
				ELSE
					sLine	:=	fbFileGets.sLine; //store line
					IF RIGHT(sLine,1) = '$L' THEN
						sLine	:=	REPLACE(sLINE, '$R$L', 2, LEN(sLine)); //restore CRLF characters
					END_IF
					Step	:=	Step + 1;
				END_IF
			ELSE
				Step	:=	90;
			END_IF
		ELSE
			Step	:=	3;
		END_IF
	END_IF
	
5:	//Parse line
	
	fbReader.eCmd	:=	eEnumCmd_First;	//Read first value (temperature)
	fbReader(pBuffer:=ADR(sLine), cbBuffer:=SIZEOF(sLine));
	
	IF fbReader.bOk THEN
		TempConvDat.VR10[nLine-1,2] := STRING_TO_REAL(fbReader.getValue);	//account for header
	ELSE
		Step	:=	90;
	END_IF	
	
	fbReader.eCmd	:=	eEnumCmd_Next;	//Read next value (resistance)
	fbReader(pBuffer:=ADR(sLine), cbBuffer:=SIZEOF(sLine));
	
	IF fbReader.bOk THEN
		TempConvDat.VR10[nLine-1,1] := STRING_TO_REAL(fbReader.getValue); //account for header
	ELSE
		Step	:=	90;
	END_IF
	
	//Read next line
	Step	:=	3;
	
10:	//end of csv file
	IF (hFile <> 0) THEN
		Step	:=	20; //close file
	END_IF
	
20:	//close csv file
	fbFileClose(bExecute:=FALSE);
	fbFileClose(sNetId:='', hFile:=hFile, bExecute:=TRUE, tTimeout:=T#5S);
	Step	:=	21;
	
21:	
	fbFileClose(bExecute:=FALSE);
	IF NOT fbFileClose.bBusy THEN
		step	:=	0;	//Standby mode
		bCompleted	:=	TRUE;
	END_IF
	
90:	//TODO: Error handling
	bError	:=	TRUE;
	IF (hFile <> 0) THEN
		Step	:=	20;	//close file
	END_IF

END_CASE

END_FUNCTION_BLOCK

// ---- POUs/Initialize/FB_InitTimes.TcPOU
FUNCTION_BLOCK FB_InitTimes
VAR_INPUT
END_VAR
VAR_OUTPUT
	bReady				:	BOOL := False;
END_VAR
VAR
	SysTim				:	NT_GetTime;
	dtCurTime			:	DT;
END_VAR

IF SysTim.BUSY THEN
	SysTim(Start:=FALSE);
ELSE
	SysTim(NetID:='', Start:=TRUE);
END_IF

IF NOT SysTim.BUSY THEN
	dtCurTime	:=	SYSTEMTIME_TO_DT(SysTim.TIMESTR);
	StateMachine.dtLastStart	:=	dtCurTime;
	StateMachine.dtLastStop		:=	dtCurTime;
	bReady	:= TRUE;
END_IF

END_FUNCTION_BLOCK

// ---- POUs/MAIN.TcPOU
PROGRAM MAIN
VAR
END_VAR

//MAIN PROGRAM

//State machine
CASE StateMachine.eStatus OF
	
	Initialize:		//Read sensor data from csv files
		P_InitMain();
		P_GetTime();
		
		IF P_InitMain.bError THEN //Initialization failed
			StateMachine.bFault		:=	TRUE;
			StateMachine.nFault		:=	10;
			StateMachine.sFaultMess	:=	'Initialization failed';
			StateMachine.eStatus	:=	Error;
		END_IF
		
		IF P_InitMain.bComplete THEN
			StateMachine.eStatus	:=	Read;
		END_IF

	Read:			//Read data from terminals and convert to physical values
		P_ReadMain();
		P_GetTime();
		StateMachine.eStatus	:=	SystemCheck;
		
		//%%%%%%%%%%%%%%%%%%%%%%%%%%%%%%%%%%%%%%%%%%%%%%%%%%%%%%%%%%%%%%%%%%%%%%%%%%%%%%%%%%%%%%%%%%%%%%%%%%%%%%%%%%%%%%%%%%%%%%%%%%%%%%%%%%%%%
		//P_TestVals();	//only for testing purposes
		//%%%%%%%%%%%%%%%%%%%%%%%%%%%%%%%%%%%%%%%%%%%%%%%%%%%%%%%%%%%%%%%%%%%%%%%%%%%%%%%%%%%%%%%%%%%%%%%%%%%%%%%%%%%%%%%%%%%%%%%%%%%%%%%%%%%%%
		
	SystemCheck:	//Check system
		P_SysCheckMain();
		IF StateMachine.bFault THEN
			StateMachine.nErrCount	:=	StateMachine.nErrCount + 1;
			P_WriteErrLog(bStart:=TRUE);			//Start writing error log
			StateMachine.eStatus	:=	Error;		//Error handling
		ELSE
			StateMachine.eStatus	:=	Automatic;	//Control
		END_IF
	
	Automatic:		//Automatic heat pump control
		P_ControlMain(bEmOp:=FALSE);
		StateMachine.eStatus	:=	Write;
		
		IF StateMachine.bManEmShutdown THEN
			StateMachine.eStatus	:=	Error;	//switch to error mode to execute emergency shutdown
		END_IF
	
	Write:			//Write control signals to terminal
		P_WriteMain();
		StateMachine.eStatus	:=	Read;
	
	Error:			//Error handling
		
		IF NOT StateMachine.bEmOpAct THEN
			P_EmShutdownMain();		//execute emergency shutdowns
		END_IF
		
		P_ErrorHandlingMain();	//execute error handling
		
		P_GetTime();			//update time
		P_WriteErrLog(bStart:=FALSE);	//finish writing error log
		
		IF StateMachine.bTempShut AND (NOT StateMachine.bPermShut) THEN	//temporary shutdown
			P_ReadMain();		//read terminals
			//%%%%%%%%%%%%%%%%%%%%%%%%%%%%%%%%%%%%%%%%%%%%%%%%%%%%%%%%%%%%%%%%%%%%%%%%%%%%%%%%%%%%%%%%%%%%%%%%%%%%%%%%%%%%%%%%%%%%%%%%%%%%%%%%%%%%%
			//P_TestVals();	//only for testing purposes
			//%%%%%%%%%%%%%%%%%%%%%%%%%%%%%%%%%%%%%%%%%%%%%%%%%%%%%%%%%%%%%%%%%%%%%%%%%%%%%%%%%%%%%%%%%%%%%%%%%%%%%%%%%%%%%%%%%%%%%%%%%%%%%%%%%%%%%
			P_SysCheckMain();	//execute system check
			IF (NOT (SysCheck.bAmbTemp OR SysCheck.bBP OR SysCheck.bCompCyc OR SysCheck.bCompOut OR SysCheck.bHCP OR 
				SysCheck.bHeatTemp OR SysCheck.bPhaseSeqCh OR SysCheck.bSensErr OR SysCheck.bTermErrRT)) THEN
				//no faults any more -> restart system
				StateMachine.bTempShut	:=	FALSE;
				StateMachine.bEmOpAct	:=	FALSE;
				StateMachine.bEmOpPoss	:=	FALSE;
				StateMachine.bFault		:=	FALSE;
				StateMachine.nFault		:=	0;
				StateMachine.sFaultMess	:=	'';
				StateMachine.eStatus	:=	Read;
			ELSE
				StateMachine.eStatus	:=	Error;	//stay in error state
			END_IF
		ELSIF StateMachine.bPermShut THEN	//permanent shutdown
				StateMachine.eStatus	:=	Error;	//stay in error state
		END_IF
		
		IF StateMachine.bEmOpPoss AND StateMachine.bActAuxHeat THEN	//emergency operation
			StateMachine.bEmOpAct	:=	TRUE;
			P_ControlMain(bEmOp:=TRUE);			//emergency operation control
			P_WriteMain();						//write values for emergency operation
		ELSE
			StateMachine.bEmOpAct	:=	FALSE;
		END_IF

END_CASE

END_PROGRAM

// ---- POUs/P_GetTime.TcPOU
PROGRAM P_GetTime
VAR
	SysTim		:	NT_GetTime;
END_VAR

IF SysTim.BUSY THEN
	SysTim(Start:=FALSE);
ELSE
	StateMachine.dtCurTime	:=	SYSTEMTIME_TO_DT(SysTim.TIMESTR);
	SysTim(Start:=FALSE);
	SysTim(Start:=TRUE);
	StateMachine.todCurTime	:=	DT_TO_TOD(StateMachine.dtCurTime);
END_IF

END_PROGRAM

// ---- POUs/Read/F_NTCSens.TcPOU
FUNCTION F_NTCSens : ST_InputVar
VAR_INPUT
	stInput	:	ST_InputVar;
	pIntTab	:	POINTER TO ARRAY[1..40,1..2] OF REAL;	//pointer to interpolation table
END_VAR
VAR
	IntTab		:	ARRAY[1..40,1..2] OF REAL;
	i			:	INT	:= 1;
	nIntElem	:	REAL;
	nLeftInd	:	INT;
	nRightInd	:	INT;
	bFound		:	BOOL	:=	FALSE;	//flag if left and right element were found
END_VAR

IntTab		:=	pIntTab^; //get interpolation table
nIntElem	:=	DINT_TO_REAL(stInput.nVarInput);
//search left and right element in interpolation table
(*
negative temperature coefficient -> table gradient is negative at all time
=> search for first element smaller than the interpolation element
*)
FOR i:=1 TO 40 DO
	IF NOT bFound THEN	
		IF (IntTab[i,1] <= nIntElem) THEN
			nRightInd	:= i;
			nLeftInd	:= i-1;
			bFound	:=	TRUE;
		END_IF
	END_IF
END_FOR

IF (NOT bFound) OR (nLeftInd < 1) THEN	//check for valid range
	stInput.bValid	:=	FALSE;	//value could not be found in interpolation table
ELSE	//perform interpolation
	stInput.fVal	:=	IntTab[nLeftInd,2] + ((nIntElem - IntTab[nLeftInd,1])/(IntTab[nRightInd,1] - IntTab[nLeftInd,1])) * (IntTab[nRightInd,2] - IntTab[nLeftInd,2]);
END_IF

IF stInput.bSensErr THEN	//check if sensor value is valid
	stInput.bValid	:=	FALSE;
END_IF

//output
F_NTCSens	:= stInput;

END_FUNCTION

// ---- POUs/Read/F_PowMeasPhase.TcPOU
FUNCTION F_PowMeasPhase : ST_InputVar_PowMeas
VAR_INPUT
	stInput	:	ST_InputVar_PowMeas;
END_VAR
VAR
END_VAR

stInput.fCurrent	:=	DINT_TO_REAL(stInput.nCurrentRaw) * stInput.fScaleCurr * stInput.fCurrTrans;	//current
stInput.fVolt		:=	DINT_TO_REAL(stInput.nVoltRaw) * stInput.fScaleVolt;							//volt
stInput.fEffPow		:=	DINT_TO_REAL(stInput.nEffPowRaw) * stInput.fScaleEffPow * stInput.fCurrTrans;	//effective power
stInput.fcosPhi		:=	DINT_TO_REAL(stInput.nVariantRaw) * stInput.fScaleCosPhi;						//power factor

END_FUNCTION

// ---- POUs/Read/P_TestVals.TcPOU
PROGRAM P_TestVals
VAR
	eVR10	:	E_TempSensVR10;
	eVR11	:	E_TempSensVR11;
	ePT100	:	E_TempSensPT100;
	ePress	:	E_Press;
END_VAR

//Manually set appropriate values
for eVR10:=SP to RF1 do
	Temperatures.stTempSensVR10[eVR10].bValid	:=	TRUE;
END_FOR

FOR eVR11:=T1 TO T8 DO
	Temperatures.stTempSensVR11[eVR11].bValid	:=	TRUE;
END_FOR

FOR ePT100:=TExpVEv TO TAmb DO
	Temperatures.stTempSensPT100[ePT100].bValid	:=	TRUE;
END_FOR

FOR ePress:=HP TO BP DO
	Pressures.stPress[ePress].bValid			:=	TRUE;
END_FOR

ePress	:=	LP;
Pressures.stPress[ePress].fVal	:=	3;
ePress	:=	HP;
Pressures.stPress[ePress].fVal	:=	25;
ePress	:=	BP;
Pressures.stPress[ePress].fVal	:=	2;
ePress	:=	HCP;
Pressures.stPress[ePress].fVal	:=	5;

END_PROGRAM

// ---- POUs/SystemCheck/F_CheckAmbTemp.TcPOU
FUNCTION F_CheckAmbTemp : BOOL
VAR_INPUT
END_VAR
VAR
	eAmbTemp	:	E_TempSensPT100 :=	TAmb;
	
	bAmbTempF	:	BOOL	:=	FALSE;
END_VAR

bAmbTempF	:=	FALSE;

//check ambient temperature
IF Temperatures.stTempSensPT100[eAmbTemp].fVal > SysCheckParams.fMaxAmbTemp THEN
	bAmbTempF				:=	TRUE;
	StateMachine.bFault		:=	TRUE;
	StateMachine.nFault		:=	41;
	StateMachine.sFaultMess	:=	'Ambient temperature too high';
END_IF

IF Temperatures.stTempSensPT100[eAmbTemp].fVal < SysCheckParams.fMinAmbTemp THEN
	bAmbTempF				:=	TRUE;
	StateMachine.bFault		:=	TRUE;
	StateMachine.nFault		:=	42;
	StateMachine.sFaultMess	:=	'Ambient temperature too low';
END_IF

IF (Temperatures.stTempSensPT100[eAmbTemp].fVal < (SysCheckParams.fMaxAmbTemp - 1)) AND 
		(Temperatures.stTempSensPT100[eAmbTemp].fVal > (SysCheckParams.fMinAmbTemp + 1)) THEN
	bAmbTempF	:=	FALSE;
END_IF

//assign output
F_CheckAmbTemp	:=	bAmbTempF;

END_FUNCTION

// ---- POUs/SystemCheck/F_CheckBrinePressure.TcPOU
FUNCTION F_CheckBrinePressure : BOOL
VAR_INPUT
END_VAR
VAR
	eBP				:	E_Press	:=	BP;	
	bBrinePressF	:	BOOL	:=	FALSE;
END_VAR

//check brine pressure
IF Pressures.stPress[eBP].fVal < SysCheckParams.fBPMinOff THEN
	bBrinePressF			:=	TRUE;
	StateMachine.bFault		:=	TRUE;
	StateMachine.nFault		:=	43;
	StateMachine.sFaultMess	:=	'Brine pressure too low';
END_IF

IF Pressures.stPress[eBP].fVal > SysCheckParams.fBPMinOn THEN
	bBrinePressF			:=	FALSE;
	(*
	Do not reset StateMachine fault here, in case there are other system faults!
	*)
END_IF

//assign output
F_CheckBrinePressure	:=	bBrinePressF;

END_FUNCTION

// ---- POUs/SystemCheck/F_CheckHeatCirTemp.TcPOU
FUNCTION F_CheckHeatCirTemp : BOOL
VAR_INPUT
END_VAR
VAR
	eT5					:	E_TempSensVR11	:=	T5;
	eT6					:	E_TempSensVR11	:=	T6;
	bHeatCirTempF		:	BOOL	:=	FALSE;
END_VAR

bHeatCirTempF	:=	FALSE;

//check heating circuit temperatures
IF Temperatures.stTempSensVR11[eT5].fVal > SysCheckParams.fTempHeatRetMax THEN
	bHeatCirTempF			:=	TRUE;
	StateMachine.bFault		:=	TRUE;
	StateMachine.nFault		:=	31;
	StateMachine.sFaultMess	:=	'Water return temperature too high';
END_IF

IF Temperatures.stTempSensVR11[eT6].fVal > SysCheckParams.fTempHeatSuppMax THEN
	bHeatCirTempF			:=	TRUE;
	StateMachine.bFault		:=	TRUE;
	StateMachine.nFault		:=	32;
	StateMachine.sFaultMess	:=	'Water supply temperature too high';
END_IF

IF (Temperatures.stTempSensVR11[eT5].fVal < (SysCheckParams.fTempHeatRetMax - 2)) 
		AND (Temperatures.stTempSensVR11[eT6].fVal < (SysCheckParams.fTempHeatSuppMax -2)) THEN
	bHeatCirTempF	:=	FALSE;
END_IF

//assign output
F_CheckHeatCirTemp	:=	bHeatCirTempF;

END_FUNCTION

// ---- POUs/SystemCheck/F_CheckPhaseSeq.TcPOU
FUNCTION F_CheckPhaseSeq : BOOL
VAR_INPUT
END_VAR
VAR
	bPhaseSeqF	:	BOOL	:=	FALSE;
END_VAR

bPhaseSeqF	:=	FALSE;

//Check phase sequence
IF PowMeas.bPhaseSeq THEN
	bPhaseSeqF				:=	TRUE;
	StateMachine.bFault		:=	TRUE;
	StateMachine.nFault		:=	47;
	StateMachine.sFaultMess	:=	'Wrong phase sequence detected';
END_IF

//assign output
F_CheckPhaseSeq :=	bPhaseSeqF;

END_FUNCTION

// ---- POUs/SystemCheck/F_CheckSens.TcPOU
FUNCTION F_CheckSens : BOOL
VAR_INPUT
END_VAR
VAR
	eTempVR10	:	E_TempSensVR10;
	eTempVR11	:	E_TempSensVR11;
	eTempPT100	:	E_TempSensPT100;
	ePress		:	E_Press;
	
	bSensErr	:	BOOL	:=	False;
END_VAR

bSensErr	:=FALSE;

//check VR10 sensors
eTempVR10	:=	SP;
IF NOT Temperatures.stTempSensVR10[eTempVR10].bValid THEN
	bSensErr				:=	TRUE;
	StateMachine.bFault		:=	TRUE;
	StateMachine.nFault		:=	81;
	StateMachine.sFaultMess	:=	'Sensor error: SP';
END_IF

eTempVR10	:=	VF1;
IF NOT Temperatures.stTempSensVR10[eTempVR10].bValid THEN
	bSensErr				:=	TRUE;
	StateMachine.bFault		:=	TRUE;
	StateMachine.nFault		:=	82;
	StateMachine.sFaultMess	:=	'Sensor error: VF1';
END_IF

eTempVR10	:=	VF2;
IF NOT Temperatures.stTempSensVR10[eTempVR10].bValid THEN
	bSensErr				:=	TRUE;
	StateMachine.bFault		:=	TRUE;
	StateMachine.nFault		:=	83;
	StateMachine.sFaultMess	:=	'Sensor error: VF2';
END_IF

eTempVR10	:=	RF1;
IF NOT Temperatures.stTempSensVR10[eTempVR10].bValid THEN
	bSensErr				:=	TRUE;
	StateMachine.bFault		:=	TRUE;
	StateMachine.nFault		:=	84;
	StateMachine.sFaultMess	:=	'Sensor error: RF1';
END_IF

//check VR11 sensors
eTempVR11	:=	T1;
IF NOT Temperatures.stTempSensVR11[eTempVR11].bValid THEN
	bSensErr				:=	TRUE;
	StateMachine.bFault		:=	TRUE;
	StateMachine.nFault		:=	71;
	StateMachine.sFaultMess	:=	'Sensor error: T1';
END_IF

eTempVR11	:=	T2;
IF NOT Temperatures.stTempSensVR11[eTempVR11].bValid THEN
	bSensErr				:=	TRUE;
	StateMachine.bFault		:=	TRUE;
	StateMachine.nFault		:=	72;
	StateMachine.sFaultMess	:=	'Sensor error: T2';
END_IF

eTempVR11	:=	T3;
IF NOT Temperatures.stTempSensVR11[eTempVR11].bValid THEN
	bSensErr				:=	TRUE;
	StateMachine.bFault		:=	TRUE;
	StateMachine.nFault		:=	73;
	StateMachine.sFaultMess	:=	'Sensor error: T3';
END_IF

eTempVR11	:=	T4;
IF NOT Temperatures.stTempSensVR11[eTempVR11].bValid THEN
	bSensErr				:=	TRUE;
	StateMachine.bFault		:=	TRUE;
	StateMachine.nFault		:=	74;
	StateMachine.sFaultMess	:=	'Sensor error: T4';
END_IF

eTempVR11	:=	T5;
IF NOT Temperatures.stTempSensVR11[eTempVR11].bValid THEN
	bSensErr				:=	TRUE;
	StateMachine.bFault		:=	TRUE;
	StateMachine.nFault		:=	75;
	StateMachine.sFaultMess	:=	'Sensor error: T5';
END_IF

eTempVR11	:=	T6;
IF NOT Temperatures.stTempSensVR11[eTempVR11].bValid THEN
	bSensErr				:=	TRUE;
	StateMachine.bFault		:=	TRUE;
	StateMachine.nFault		:=	76;
	StateMachine.sFaultMess	:=	'Sensor error: T6';
END_IF

eTempVR11	:=	T8;
IF NOT Temperatures.stTempSensVR11[eTempVR11].bValid THEN
	bSensErr				:=	TRUE;
	StateMachine.bFault		:=	TRUE;
	StateMachine.nFault		:=	78;
	StateMachine.sFaultMess	:=	'Sensor error: T8';
END_IF

//check PT100 temperature sensors 
(* 
-> additional sensors are not relevant for the system control and therefore not checked here
*)
eTempPT100	:=	TAmb;
IF NOT Temperatures.stTempSensPT100[eTempPT100].bValid THEN
	bSensErr				:=	TRUE;
	StateMachine.bFault		:=	TRUE;
	StateMachine.nFault		:=	64;
	StateMachine.sFaultMess	:=	'Sensor error: Ambient temperature';
END_IF

//check pressure sensors
ePress	:=	HP;
IF NOT Pressures.stPress[ePress].bValid THEN
	bSensErr				:=	TRUE;
	StateMachine.bFault		:=	TRUE;
	StateMachine.nFault		:=	51;
	StateMachine.sFaultMess	:=	'Sensor error: High pressure';
END_IF

ePress	:=	LP;
IF NOT Pressures.stPress[ePress].bValid THEN
	bSensErr				:=	TRUE;
	StateMachine.bFault		:=	TRUE;
	StateMachine.nFault		:=	52;
	StateMachine.sFaultMess	:=	'Sensor error: Low pressure';
END_IF

ePress	:=	HCP;
IF NOT Pressures.stPress[ePress].bValid THEN
	bSensErr				:=	TRUE;
	StateMachine.bFault		:=	TRUE;
	StateMachine.nFault		:=	53;
	StateMachine.sFaultMess	:=	'Sensor error: Heating circuit pressure';
END_IF

ePress	:=	BP;
IF NOT Pressures.stPress[ePress].bValid THEN
	bSensErr				:=	TRUE;
	StateMachine.bFault		:=	TRUE;
	StateMachine.nFault		:=	54;
	StateMachine.sFaultMess	:=	'Sensor error: Brine pressure';
END_IF

//Assign output
F_CheckSens	:=	bSensErr;

END_FUNCTION

// ---- POUs/SystemCheck/F_CheckTerm.TcPOU
FUNCTION F_CheckTerm : BOOL
VAR_INPUT
END_VAR
VAR
	eTerm		:	E_Terminals;

	bTermErr	:	BOOL	:=	FALSE;
END_VAR

bTermErr	:=	FALSE;

//Check all terminals
eTerm	:=	TempSens1;
IF TerminalErrorRT.bTermRt[eTerm] THEN
	bTermErr			:=	TRUE;
	StateMachine.bFault	:=	TRUE;
	StateMachine.nFault	:=	91;
	StateMachine.sFaultMess	:=	'Real-time communication with terminal failed: TempSens1';
END_IF

eTerm	:=	TempSens2;
IF TerminalErrorRT.bTermRt[eTerm] THEN
	bTermErr			:=	TRUE;
	StateMachine.bFault	:=	TRUE;
	StateMachine.nFault	:=	92;
	StateMachine.sFaultMess	:=	'Real-time communication with terminal failed: TempSens2';
END_IF

eTerm	:=	TempSens3;
IF TerminalErrorRT.bTermRt[eTerm] THEN
	bTermErr			:=	TRUE;
	StateMachine.bFault	:=	TRUE;
	StateMachine.nFault	:=	93;
	StateMachine.sFaultMess	:=	'Real-time communication with terminal failed: TempSens3';
END_IF

eTerm	:=	TempSens3Wire;
IF TerminalErrorRT.bTermRt[eTerm] THEN
	bTermErr			:=	TRUE;
	StateMachine.bFault	:=	TRUE;
	StateMachine.nFault	:=	94;
	StateMachine.sFaultMess	:=	'Real-time communication with terminal failed: TempSens3Wire';
END_IF

eTerm	:=	PressSens;
IF TerminalErrorRT.bTermRt[eTerm] THEN
	bTermErr			:=	TRUE;
	StateMachine.bFault	:=	TRUE;
	StateMachine.nFault	:=	95;
	StateMachine.sFaultMess	:=	'Real-time communication with terminal failed: PressSens';
END_IF

eTerm	:=	PowMeasTerm;
IF TerminalErrorRT.bTermRt[eTerm] THEN
	bTermErr			:=	TRUE;
	StateMachine.bFault	:=	TRUE;
	StateMachine.nFault	:=	96;
	StateMachine.sFaultMess	:=	'Real-time communication with terminal failed: PowMeas';
END_IF

eTerm	:=	AnalogOutp;
IF TerminalErrorRT.bTermRt[eTerm] THEN
	bTermErr			:=	TRUE;
	StateMachine.bFault	:=	TRUE;
	StateMachine.nFault	:=	97;
	StateMachine.sFaultMess	:=	'Real-time communication with terminal failed: AnalogOutp';
END_IF

eTerm	:=	OutpSwitchValv;
IF TerminalErrorRT.bTermRt[eTerm] THEN
	bTermErr			:=	TRUE;
	StateMachine.bFault	:=	TRUE;
	StateMachine.nFault	:=	98;
	StateMachine.sFaultMess	:=	'Real-time communication with terminal failed: OutpSwitchValv';
END_IF

eTerm	:=	OutpCont;
IF TerminalErrorRT.bTermRt[eTerm] THEN
	bTermErr			:=	TRUE;
	StateMachine.bFault	:=	TRUE;
	StateMachine.nFault	:=	99;
	StateMachine.sFaultMess	:=	'Real-time communication with terminal failed: OutpCont';
END_IF

//Assing output
F_CheckTerm	:=	bTermErr;

END_FUNCTION

// ---- POUs/Write/F_PumpConvPercVolt.TcPOU
FUNCTION F_PumpConvPercVolt : REAL
VAR_INPUT
	nPercentRPM		:	USINT;
END_VAR
VAR
	fVolt			:	REAL;
END_VAR

//converts the relative pump rpm in percent to a voltage signal
(*
<0.5V		: cable break detection - pump runs at minimum speed (emergency operation)
0.5V - 1V	: pump stops
1V - 3V		: pump runs at minimum speed (starting)
2V - 3V		: pump runs at minimum speed (operation)
3V - 10V	: speed varies linear between minimum and maximum
*)
fVolt	:=	3 + (10 - 3)*(USINT_TO_SINT(nPercentRPM)/100);

//assign output
F_PumpConvPercVolt	:=	fVolt;

END_FUNCTION

// ---- POUs/Write/FB_RampPump.TcPOU
FUNCTION_BLOCK FB_RampPump
VAR_INPUT
	fStartVal	:	REAL;
	fEndVal		:	REAL;
	tDuration	:	TIME;
END_VAR
VAR_OUTPUT
	fCurVal		:	REAL;
	bActiveRamp	:	BOOL	:=	FALSE;
END_VAR
VAR
	Timer			:	TON;
	nDurMS			:	DWORD;	//duration in ms
	fInc			:	REAL;	//incremental change per ms
	nTimeAfterStart	:	DWORD;	//time after start of ramp in ms
END_VAR

IF NOT bActiveRamp THEN	//initialization
	nDurMS		:=	TIME_TO_DWORD(tDuration);
	fInc		:=	(fEndVal - fStartVal)/DWORD_TO_REAL(nDurMS);
	//reset timer
	Timer.IN	:=	FALSE;
	Timer();
	Timer.PT	:=	tDuration;
	bActiveRamp	:=	TRUE;
ELSE	//generate ramp
	Timer.IN		:=	TRUE;
	Timer();
	nTimeAfterStart	:=	TIME_TO_DWORD(Timer.ET);
	fCurVal			:=	fStartVal + fInc*DWORD_TO_REAL(nTimeAfterStart);
END_IF

IF Timer.Q THEN
	bActiveRamp	:=	FALSE;
END_IF

END_FUNCTION_BLOCK

// ---- GlobalTextList.TcGTLO
TEXTLIST GlobalTextList
  53 = '%2.1f'
  15 = '%3.2f'
  47 = '%s'
  51 = 'Activate AuxHeat'
  2 = 'Auxiliary Heater'
  35 = 'BP'
  3 = 'Brine Pump'
  6 = 'Circulating Pump'
  0 = 'Compressor'
  42 = 'Current '
  55 = 'day'
  10 = 'DHW mode'
  9 = 'DHW mode - SH mode'
  8 = 'DHW mode - Space heat mode'
  59 = 'Domestic Hot Water'
  40 = 'Effective Power '
  45 = 'Emergency Shutdown'
  5 = 'ExtHeatCir Pump'
  34 = 'HCP'
  32 = 'HP'
  4 = 'IntHeatCir Pump'
  36 = 'L1'
  37 = 'L2'
  38 = 'L3'
  33 = 'LP'
  7 = 'Manual Control'
  46 = 'Manual Emergency Shutdown'
  61 = 'max'
  60 = 'min'
  12 = 'Mixing valve position'
  56 = 'night'
  54 = 'Num. Err: %i'
  49 = 'Perm. Shutdown'
  48 = 'Permanent Shutdown'
  43 = 'Phase Error'
  41 = 'Power Factor'
  39 = 'Power Measurement'
  31 = 'Pressures'
  26 = 'RF1'
  52 = 'Room Temp.'
  58 = 'Room Temperature'
  11 = 'SHmode'
  23 = 'SP'
  44 = 'System Fault'
  16 = 'T1'
  14 = 'T1: \\t %3.2f'
  17 = 'T2'
  18 = 'T3'
  19 = 'T4'
  20 = 'T5'
  21 = 'T6'
  22 = 'T8'
  30 = 'TAmb'
  29 = 'TCond'
  50 = 'Temp. Shutdown'
  57 = 'Temperature Setpoints'
  13 = 'Temperatures'
  1 = 'Test'
  27 = 'TExpVEv'
  28 = 'TShEv'
  24 = 'VF1'
  25 = 'VF2'
END_TEXTLIST

// ---- VISUs/StandardVis.TcVIS
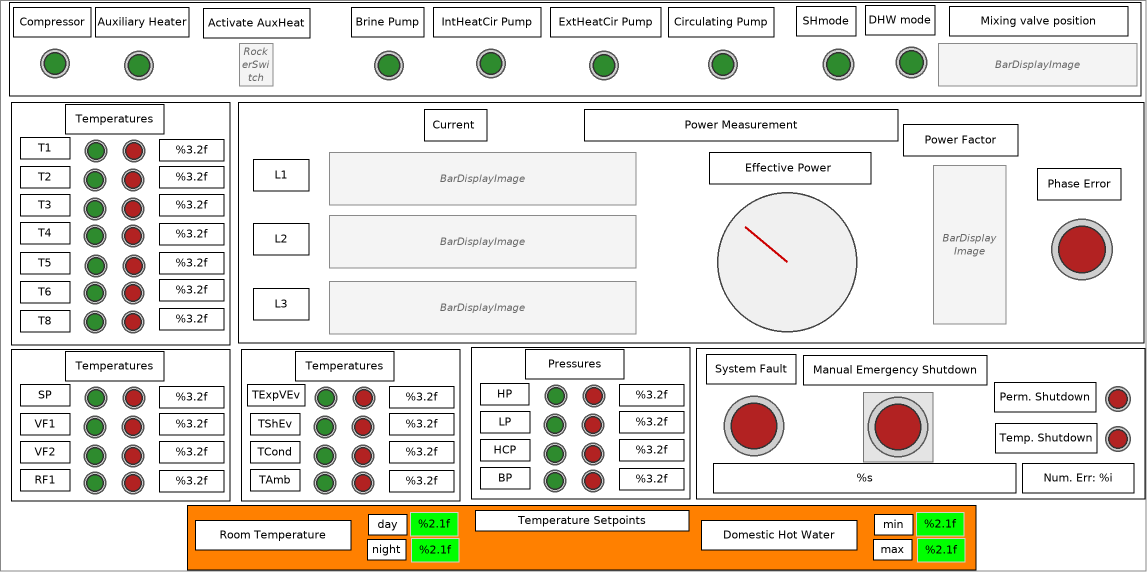
VISUALIZATION StandardVis  // 1147x572
    Group (11,102 219x243)
        Rectangle (0,0 219x243)
        Rectangle (54,2 99x30), "Temperatures"
        Rectangle (148,37 65x22), "%3.2f", text variable: Temperatures.stTempSensVR11[0].fVal
        Rectangle (148,64 65x22), "%3.2f", text variable: Temperatures.stTempSensVR11[1].fVal
        Rectangle (148,92 65x22), "%3.2f", text variable: Temperatures.stTempSensVR11[2].fVal
        Rectangle (148,121 65x22), "%3.2f", text variable: Temperatures.stTempSensVR11[3].fVal
        Rectangle (148,150 65x22), "%3.2f", text variable: Temperatures.stTempSensVR11[4].fVal
        Rectangle (148,177 65x22), "%3.2f", text variable: Temperatures.stTempSensVR11[5].fVal
        Rectangle (148,206 65x22), "%3.2f", text variable: Temperatures.stTempSensVR11[6].fVal
        Rectangle (9,35 50x22), "T1"
        Rectangle (9,64 50x22), "T2"
        Rectangle (9,92 50x22), "T3"
        Rectangle (9,120 50x22), "T4"
        Rectangle (9,150 50x22), "T5"
        Rectangle (9,179 50x22), "T6"
        Rectangle (9,208 50x22), "T8"
        Lamp1 (110,36 26x26), variable: NOT Temperatures.stTempSensVR11[0].bValid, style: Lamp-Lamp1-Red
        Lamp1 (72,36 26x26), variable: Temperatures.stTempSensVR11[0].bValid, style: Lamp-Lamp1-Green
        Lamp1 (109,65 26x26), variable: NOT Temperatures.stTempSensVR11[1].bValid, style: Lamp-Lamp1-Red
        Lamp1 (71,65 26x26), variable: Temperatures.stTempSensVR11[1].bValid, style: Lamp-Lamp1-Green
        Lamp1 (109,94 26x26), variable: NOT Temperatures.stTempSensVR11[2].bValid, style: Lamp-Lamp1-Red
        Lamp1 (71,94 26x26), variable: Temperatures.stTempSensVR11[2].bValid, style: Lamp-Lamp1-Green
        Lamp1 (109,121 26x26), variable: NOT Temperatures.stTempSensVR11[3].bValid, style: Lamp-Lamp1-Red
        Lamp1 (71,121 26x26), variable: Temperatures.stTempSensVR11[3].bValid, style: Lamp-Lamp1-Green
        Lamp1 (110,151 26x26), variable: NOT Temperatures.stTempSensVR11[4].bValid, style: Lamp-Lamp1-Red
        Lamp1 (72,151 26x26), variable: Temperatures.stTempSensVR11[4].bValid, style: Lamp-Lamp1-Green
        Lamp1 (109,178 26x26), variable: NOT Temperatures.stTempSensVR11[5].bValid, style: Lamp-Lamp1-Red
        Lamp1 (71,178 26x26), variable: Temperatures.stTempSensVR11[5].bValid, style: Lamp-Lamp1-Green
        Lamp1 (109,207 26x26), variable: NOT Temperatures.stTempSensVR11[6].bValid, style: Lamp-Lamp1-Red
        Lamp1 (71,207 26x26), variable: Temperatures.stTempSensVR11[6].bValid, style: Lamp-Lamp1-Green
    Group (11,349 219x152)
        Rectangle (0,0 219x152)
        Rectangle (54,2 99x30), "Temperatures"
        Rectangle (148,37 65x22), "%3.2f", text variable: Temperatures.stTempSensVR10[0].fVal
        Rectangle (148,64 65x22), "%3.2f", text variable: Temperatures.stTempSensVR10[1].fVal
        Rectangle (148,92 65x22), "%3.2f", text variable: Temperatures.stTempSensVR10[2].fVal
        Rectangle (148,121 65x22), "%3.2f", text variable: Temperatures.stTempSensVR10[3].fVal
        Rectangle (9,35 50x22), "SP"
        Rectangle (9,64 50x22), "VF1"
        Rectangle (9,92 50x22), "VF2"
        Rectangle (9,120 50x22), "RF1"
        Lamp1 (110,36 26x26), variable: NOT Temperatures.stTempSensVR10[0].bValid, style: Lamp-Lamp1-Red
        Lamp1 (72,36 26x26), variable: Temperatures.stTempSensVR10[0].bValid, style: Lamp-Lamp1-Green
        Lamp1 (109,65 26x26), variable: NOT Temperatures.stTempSensVR10[1].bValid, style: Lamp-Lamp1-Red
        Lamp1 (71,65 26x26), variable: Temperatures.stTempSensVR10[1].bValid, style: Lamp-Lamp1-Green
        Lamp1 (109,94 26x26), variable: NOT Temperatures.stTempSensVR10[2].bValid, style: Lamp-Lamp1-Red
        Lamp1 (71,94 26x26), variable: Temperatures.stTempSensVR10[2].bValid, style: Lamp-Lamp1-Green
        Lamp1 (109,121 26x26), variable: NOT Temperatures.stTempSensVR10[3].bValid, style: Lamp-Lamp1-Red
        Lamp1 (71,121 26x26), variable: Temperatures.stTempSensVR10[3].bValid, style: Lamp-Lamp1-Green
    Group (241,349 219x152)
        Rectangle (0,0 219x152)
        Rectangle (54,2 99x30), "Temperatures"
        Rectangle (148,37 65x22), "%3.2f", text variable: Temperatures.stTempSensPT100[0].fVal
        Rectangle (148,64 65x22), "%3.2f", text variable: Temperatures.stTempSensPT100[1].fVal
        Rectangle (148,92 65x22), "%3.2f", text variable: Temperatures.stTempSensPT100[2].fVal
        Rectangle (148,121 65x22), "%3.2f", text variable: Temperatures.stTempSensPT100[3].fVal
        Rectangle (6,35 58x22), "TExpVEv"
        Rectangle (9,64 50x22), "TShEv"
        Rectangle (9,92 50x22), "TCond"
        Rectangle (9,120 50x22), "TAmb"
        Lamp1 (110,36 26x26), variable: NOT Temperatures.stTempSensPT100[0].bValid, style: Lamp-Lamp1-Red
        Lamp1 (72,36 26x26), variable: Temperatures.stTempSensPT100[0].bValid, style: Lamp-Lamp1-Green
        Lamp1 (109,65 26x26), variable: NOT Temperatures.stTempSensPT100[1].bValid, style: Lamp-Lamp1-Red
        Lamp1 (71,65 26x26), variable: Temperatures.stTempSensPT100[1].bValid, style: Lamp-Lamp1-Green
        Lamp1 (109,94 26x26), variable: NOT Temperatures.stTempSensPT100[2].bValid, style: Lamp-Lamp1-Red
        Lamp1 (71,94 26x26), variable: Temperatures.stTempSensPT100[2].bValid, style: Lamp-Lamp1-Green
        Lamp1 (109,121 26x26), variable: NOT Temperatures.stTempSensPT100[3].bValid, style: Lamp-Lamp1-Red
        Lamp1 (71,121 26x26), variable: Temperatures.stTempSensPT100[3].bValid, style: Lamp-Lamp1-Green
    Group (471,347 219x152)
        Rectangle (0,0 219x152)
        Rectangle (54,2 99x30), "Pressures"
        Rectangle (148,37 65x22), "%3.2f", text variable: Pressures.stPress[0].fVal
        Rectangle (148,64 65x22), "%3.2f", text variable: Pressures.stPress[1].fVal
        Rectangle (148,92 65x22), "%3.2f", text variable: Pressures.stPress[2].fVal
        Rectangle (148,121 65x22), "%3.2f", text variable: Pressures.stPress[3].fVal
        Rectangle (9,36 49x22), "HP"
        Rectangle (9,64 50x22), "LP"
        Rectangle (9,92 50x22), "HCP"
        Rectangle (9,120 50x22), "BP"
        Lamp1 (110,36 26x26), variable: NOT Pressures.stPress[0].bValid, style: Lamp-Lamp1-Red
        Lamp1 (72,36 26x26), variable: Pressures.stPress[0].bValid, style: Lamp-Lamp1-Green
        Lamp1 (109,65 26x26), variable: NOT Pressures.stPress[1].bValid, style: Lamp-Lamp1-Red
        Lamp1 (71,65 26x26), variable: Pressures.stPress[1].bValid, style: Lamp-Lamp1-Green
        Lamp1 (109,94 26x26), variable: NOT Pressures.stPress[2].bValid, style: Lamp-Lamp1-Red
        Lamp1 (71,94 26x26), variable: Pressures.stPress[2].bValid, style: Lamp-Lamp1-Green
        Lamp1 (109,121 26x26), variable: NOT Pressures.stPress[3].bValid, style: Lamp-Lamp1-Red
        Lamp1 (71,121 26x26), variable: Pressures.stPress[3].bValid, style: Lamp-Lamp1-Green
    Group (238,102 906x241)
        Rectangle (0,0 906x241)
        BarDisplayImage (91,50 307x53), value: PowMeas.stPowMeas[0].fCurrent, style: BarDisplayImage-Gray, scale format: %.1f, scale 0..10
        BarDisplayImage (91,113 307x53), value: PowMeas.stPowMeas[1].fCurrent, style: BarDisplayImage-Gray, scale format: %.1f, scale 0..10
        BarDisplayImage (91,179 307x53), value: PowMeas.stPowMeas[2].fCurrent, style: BarDisplayImage-Gray, scale format: %.1f, scale 0..10
        Rectangle (15,57 56x32), "L1"
        Rectangle (15,121 56x32), "L2"
        Rectangle (15,186 56x32), "L3"
        Rectangle (346,7 314x32), "Power Measurement"
        Meter180 (421,90 256x140), value: PowMeas.fEffPow, style: Meter-Meter180-Gray, scale format: %.1f, scale 0..10
        Rectangle (471,50 162x32), "Effective Power"
        BarDisplayImage (695,63 73x159), value: PowMeas.fMeanCosPhi, style: BarDisplayImage-Gray, scale format: %.1f, scale 0.5..1
        Rectangle (665,22 115x32), "Power Factor"
        Rectangle (186,7 63x32), "Current"
        Rectangle (799,66 84x32), "Phase Error"
        Lamp1 (808,110 72x75), variable: PowMeas.bPhaseSeq, style: Lamp-Lamp1-Red
    Group (9,2 1132x94)
        Rectangle (0,0 1132x94)
        Rectangle (342,5 73x30), "Brine Pump"
        Lamp1 (29,41 34x41), variable: DigOutputs.bOutpComp, style: Lamp-Lamp1-Green
        Lamp1 (113,43 34x41), variable: DigOutputs.bOutpAH, style: Lamp-Lamp1-Green
        Rectangle (4,5 78x30), "Compressor"
        Rectangle (86,5 94x30), "Auxiliary Heater"
        Rectangle (424,5 108x30), "IntHeatCir Pump"
        Rectangle (541,5 111x30), "ExtHeatCir Pump"
        Rectangle (659,5 106x30), "Circulating Pump"
        Lamp1 (363,43 34x41), variable: StateMachine.bBrinePump, style: Lamp-Lamp1-Green
        Lamp1 (465,41 34x41), variable: StateMachine.bIntHeatCPump, style: Lamp-Lamp1-Green
        Lamp1 (578,43 34x41), variable: StateMachine.bExtHeatCPump, style: Lamp-Lamp1-Green
        Lamp1 (697,42 34x41), variable: StateMachine.bCircPump, style: Lamp-Lamp1-Green
        Lamp1 (804,44 51x37), variable: StateMachine.bSwitchVal, style: Lamp-Lamp1-Green
        Lamp1 (877,42 51x37), variable: NOT StateMachine.bSwitchVal, style: Lamp-Lamp1-Green
        Rectangle (856,3 70x30), "DHW mode"
        Rectangle (787,4 60x30), "SHmode"
        Rectangle (940,4 179x30), "Mixing valve position"
        BarDisplayImage (929,41 199x43), value: AnaOutputs.stOutpMixValv.fVal, style: BarDisplayImage-Gray, scale format: %.1f, scale 0..10
        Rectangle (194,6 107x30), "Activate AuxHeat"
        RockerSwitch (230,41 34x43), variable: StateMachine.bActAuxHeat, behaviour: TOGGLE, style: Switch-RockerSwitch-Blue
    Group (696,348 449x151)
        Rectangle (0,0 449x151)
        Rectangle (10,6 90x30), "System Fault"
        Lamp1 (23,43 70x70), variable: StateMachine.bFault, style: Lamp-Lamp1-Red
        Rectangle (107,7 184x30), "Manual Emergency Shutdown"
        PushSwitchLed (167,44 70x70), variable: StateMachine.bManEmShutdown, behaviour: TOGGLE, style: Switch-PushSwitchLed-Red
        Rectangle (17,115 303x30), "%s", text variable: StateMachine.sFaultMess, colour toggle: StateMachine.bFault
        Rectangle (298,34 102x30), "Perm. Shutdown"
        Rectangle (299,75 102x30), "Temp. Shutdown"
        Lamp1 (407,75 30x32), variable: StateMachine.bTempShut, style: Lamp-Lamp1-Red
        Lamp1 (407,35 30x32), variable: StateMachine.bPermShut, style: Lamp-Lamp1-Red
        Rectangle (326,115 112x30), "Num. Err: %i", text variable: StateMachine.nErrCount
    Group (187,505 789x65)
        Rectangle (0,0 789x65)
        Rectangle (288,5 214x21), "Temperature Setpoints"
        Rectangle (8,15 156x30), "Room Temperature"
        Textfield (223,7 48x24), "%2.1f", text variable: TempSetpoints.fRoomSetpoint, input disabled if: FALSE
            OnMouseClick: write the text variable via VisuDialogs.Numpad, min 5, max 25
        Textfield (224,33 48x24), "%2.1f", text variable: TempSetpoints.fRoomSetpointNight, input disabled if: FALSE
            OnMouseClick: write the text variable via VisuDialogs.Numpad, min 5, max 25
        Rectangle (181,9 39x21), "day"
        Rectangle (180,34 39x21), "night"
        Rectangle (514,15 156x30), "Domestic Hot Water"
        Textfield (729,7 48x24), "%2.1f", text variable: TempSetpoints.fDHWLowSP, input disabled if: FALSE
            OnMouseClick: write the text variable via VisuDialogs.Numpad, min 30, max TempSetpoints.fDHWUpSP - 1
        Textfield (730,33 48x24), "%2.1f", text variable: TempSetpoints.fDHWUpSP, input disabled if: FALSE
            OnMouseClick: write the text variable via VisuDialogs.Numpad, min TempSetpoints.fDHWLowSP + 1, max 70
        Rectangle (687,9 39x21), "min"
        Rectangle (686,34 39x21), "max"
END_VISUALIZATION
